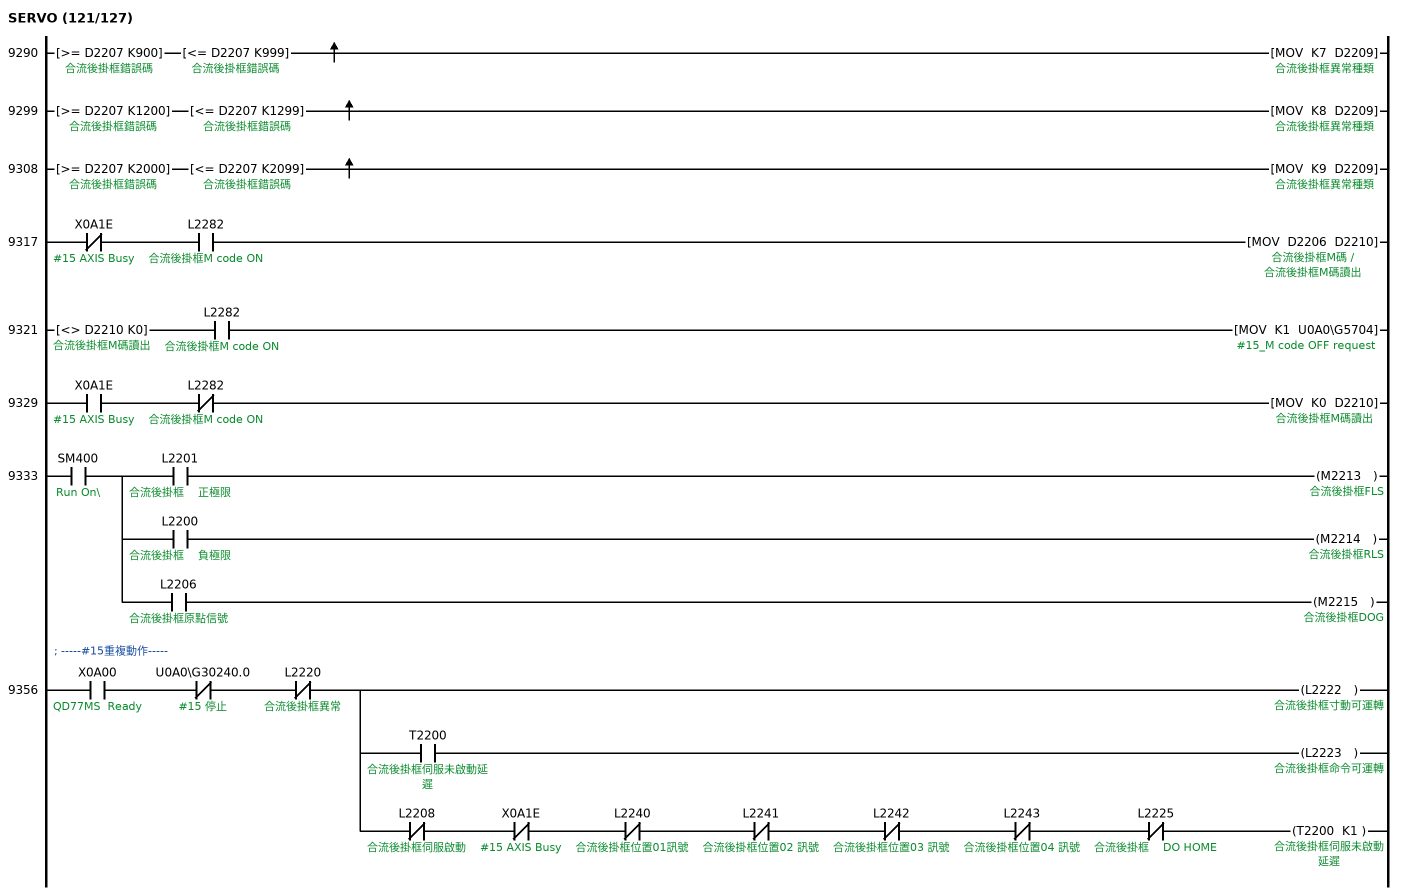
[picture p120: ladder of SERVO, rungs at steps 9290 to 9356]
9290  LD>=    D2207 K900  ; 合流後掛框錯誤碼
      AND<=   D2207 K999  ; 合流後掛框錯誤碼
      MEP
      MOV     K7 D2209
9299  LD>=    D2207 K1200  ; 合流後掛框錯誤碼
      AND<=   D2207 K1299  ; 合流後掛框錯誤碼
      MEP
      MOV     K8 D2209
9308  LD>=    D2207 K2000  ; 合流後掛框錯誤碼
      AND<=   D2207 K2099  ; 合流後掛框錯誤碼
      MEP
      MOV     K9 D2209
9317  LDI     X0A1E  ; #15 AXIS Busy
      AND     L2282  ; 合流後掛框M code ON
      MOV     D2206 D2210  ; 合流後掛框M碼讀出
9321  LD<>    D2210 K0  ; 合流後掛框M碼讀出
      AND     L2282  ; 合流後掛框M code ON
      MOV     K1 U0A0\G5704  ; #15_M code OFF request
9329  LD      X0A1E  ; #15 AXIS Busy
      ANI     L2282  ; 合流後掛框M code ON
      MOV     K0 D2210
9333  LD      SM400  ; Run On\
      MPS
      AND     L2201  ; 合流後掛框    正極限
      OUT     M2213  ; 合流後掛框FLS
      MRD
      AND     L2200  ; 合流後掛框    負極限
      OUT     M2214  ; 合流後掛框RLS
      MPP
      AND     L2206  ; 合流後掛框原點信號
      OUT     M2215  ; 合流後掛框DOG
; -----#15重複動作-----
9356  LD      X0A00  ; QD77MS  Ready
      ANI     U0A0\G30240.0  ; #15 停止
      ANI     L2220  ; 合流後掛框異常
      OUT     L2222  ; 合流後掛框寸動可運轉
      MPS
      AND     T2200  ; 合流後掛框伺服未啟動延遲
      OUT     L2223  ; 合流後掛框命令可運轉
      MPP
      ANI     L2208  ; 合流後掛框伺服啟動
      ANI     X0A1E  ; #15 AXIS Busy
      ANI     L2240  ; 合流後掛框位置01訊號
      ANI     L2241  ; 合流後掛框位置02 訊號
      ANI     L2242  ; 合流後掛框位置03 訊號
      ANI     L2243  ; 合流後掛框位置04 訊號
      ANI     L2225  ; 合流後掛框    DO HOME
      OUT     T2200 K1  ; 合流後掛框伺服未啟動延遲
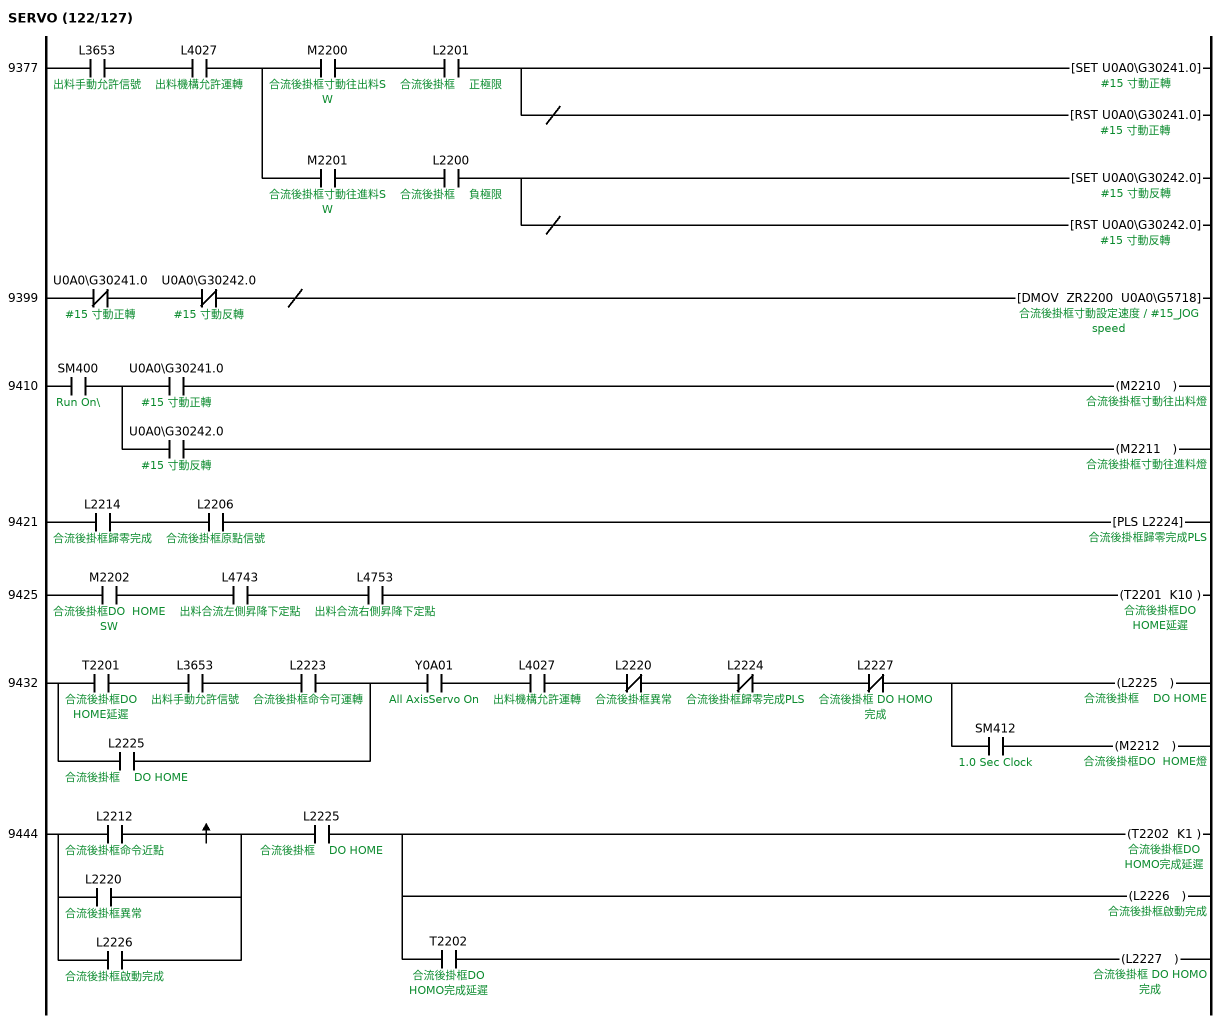
9377  LD      L3653  ; 出料手動允許信號
      AND     L4027  ; 出料機構允許運轉
      MPS
      AND     M2200  ; 合流後掛框寸動往出料SW
      AND     L2201  ; 合流後掛框    正極限
      SET     U0A0\G30241.0  ; #15 寸動正轉
      INV
      RST     U0A0\G30241.0  ; #15 寸動正轉
      MPP
      AND     M2201  ; 合流後掛框寸動往進料SW
      AND     L2200  ; 合流後掛框    負極限
      SET     U0A0\G30242.0  ; #15 寸動反轉
      INV
      RST     U0A0\G30242.0  ; #15 寸動反轉
9399  LDI     U0A0\G30241.0  ; #15 寸動正轉
      ANI     U0A0\G30242.0  ; #15 寸動反轉
      INV
      DMOV    ZR2200 U0A0\G5718  ; 合流後掛框寸動設定速度 / #15_JOG     speed
9410  LD      SM400  ; Run On\
      MPS
      AND     U0A0\G30241.0  ; #15 寸動正轉
      OUT     M2210  ; 合流後掛框寸動往出料燈
      MPP
      AND     U0A0\G30242.0  ; #15 寸動反轉
      OUT     M2211  ; 合流後掛框寸動往進料燈
9421  LD      L2214  ; 合流後掛框歸零完成
      AND     L2206  ; 合流後掛框原點信號
      PLS     L2224  ; 合流後掛框歸零完成PLS
9425  LD      M2202  ; 合流後掛框DO  HOME SW
      AND     L4743  ; 出料合流左側昇降下定點
      AND     L4753  ; 出料合流右側昇降下定點
      OUT     T2201 K10  ; 合流後掛框DO HOME延遲
9432  LD      T2201  ; 合流後掛框DO HOME延遲
      AND     L3653  ; 出料手動允許信號
      AND     L2223  ; 合流後掛框命令可運轉
      OR      L2225  ; 合流後掛框    DO HOME
      AND     Y0A01  ; All AxisServo On
      AND     L4027  ; 出料機構允許運轉
      ANI     L2220  ; 合流後掛框異常
      ANI     L2224  ; 合流後掛框歸零完成PLS
      ANI     L2227  ; 合流後掛框 DO HOMO 完成
      OUT     L2225  ; 合流後掛框    DO HOME
      AND     SM412  ; 1.0 Sec Clock
      OUT     M2212  ; 合流後掛框DO  HOME燈
9444  LD      L2212  ; 合流後掛框命令近點
      MEP
      OR      L2220  ; 合流後掛框異常
      OR      L2226  ; 合流後掛框啟動完成
      AND     L2225  ; 合流後掛框    DO HOME
      OUT     T2202 K1  ; 合流後掛框DO HOMO完成延遲
      OUT     L2226  ; 合流後掛框啟動完成
      AND     T2202  ; 合流後掛框DO HOMO完成延遲
      OUT     L2227  ; 合流後掛框 DO HOMO 完成
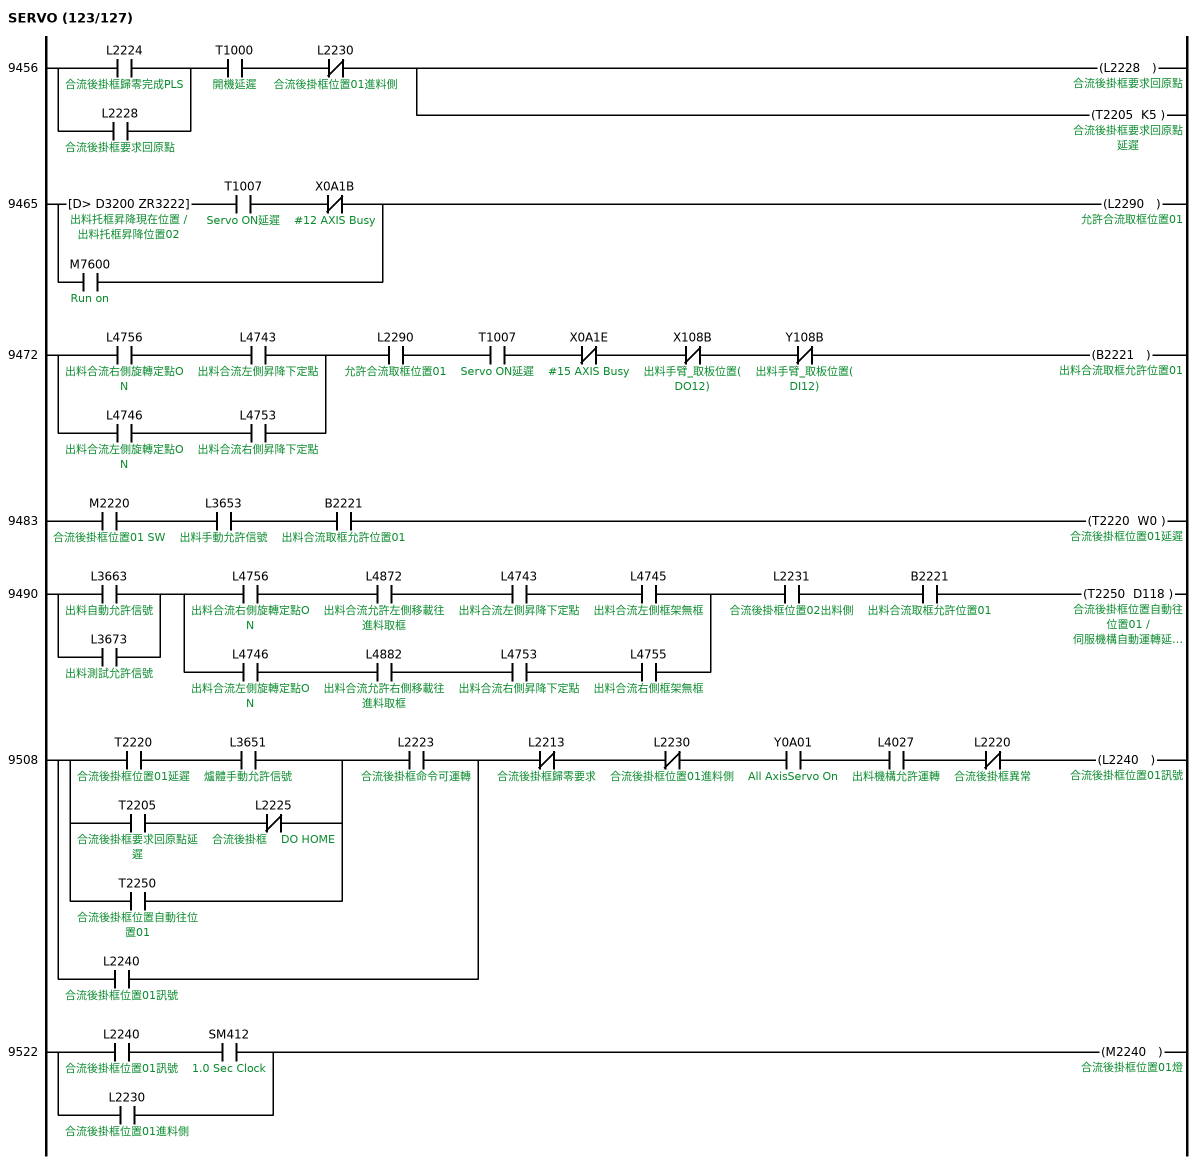
9456  LD      L2224  ; 合流後掛框歸零完成PLS
      OR      L2228  ; 合流後掛框要求回原點
      AND     T1000  ; 開機延遲
      ANI     L2230  ; 合流後掛框位置01進料側
      OUT     L2228  ; 合流後掛框要求回原點
      OUT     T2205 K5  ; 合流後掛框要求回原點延遲
9465  LDD>    D3200 ZR3222  ; 出料托框昇降現在位置 / 出料托框昇降位置02
      AND     T1007  ; Servo ON延遲
      ANI     X0A1B  ; #12 AXIS Busy
      OR      M7600  ; Run on
      OUT     L2290  ; 允許合流取框位置01
9472  LD      L4756  ; 出料合流右側旋轉定點ON
      AND     L4743  ; 出料合流左側昇降下定點
      LD      L4746  ; 出料合流左側旋轉定點ON
      AND     L4753  ; 出料合流右側昇降下定點
      ORB
      AND     L2290  ; 允許合流取框位置01
      AND     T1007  ; Servo ON延遲
      ANI     X0A1E  ; #15 AXIS Busy
      ANI     X108B  ; 出料手臂_取板位置(DO12)
      ANI     Y108B  ; 出料手臂_取板位置(DI12)
      OUT     B2221  ; 出料合流取框允許位置01
9483  LD      M2220  ; 合流後掛框位置01 SW
      AND     L3653  ; 出料手動允許信號
      AND     B2221  ; 出料合流取框允許位置01
      OUT     T2220 W0  ; 合流後掛框位置01延遲
9490  LD      L3663  ; 出料自動允許信號
      OR      L3673  ; 出料測試允許信號
      LD      L4756  ; 出料合流右側旋轉定點ON
      AND     L4872  ; 出料合流允許左側移載往  進料取框
      AND     L4743  ; 出料合流左側昇降下定點
      AND     L4745  ; 出料合流左側框架無框
      LD      L4746  ; 出料合流左側旋轉定點ON
      AND     L4882  ; 出料合流允許右側移載往  進料取框
      AND     L4753  ; 出料合流右側昇降下定點
      AND     L4755  ; 出料合流右側框架無框
      ORB
      ANB
      AND     L2231  ; 合流後掛框位置02出料側
      AND     B2221  ; 出料合流取框允許位置01
      OUT     T2250 D118  ; 合流後掛框位置自動往位置01 / 伺服機構自動運轉延遲時間
9508  LD      T2220  ; 合流後掛框位置01延遲
      AND     L3651  ; 爐體手動允許信號
      LD      T2205  ; 合流後掛框要求回原點延遲
      ANI     L2225  ; 合流後掛框    DO HOME
      ORB
      OR      T2250  ; 合流後掛框位置自動往位置01
      AND     L2223  ; 合流後掛框命令可運轉
      OR      L2240  ; 合流後掛框位置01訊號
      ANI     L2213  ; 合流後掛框歸零要求
      ANI     L2230  ; 合流後掛框位置01進料側
      AND     Y0A01  ; All AxisServo On
      AND     L4027  ; 出料機構允許運轉
      ANI     L2220  ; 合流後掛框異常
      OUT     L2240  ; 合流後掛框位置01訊號
9522  LD      L2240  ; 合流後掛框位置01訊號
      AND     SM412  ; 1.0 Sec Clock
      OR      L2230  ; 合流後掛框位置01進料側
      OUT     M2240  ; 合流後掛框位置01燈
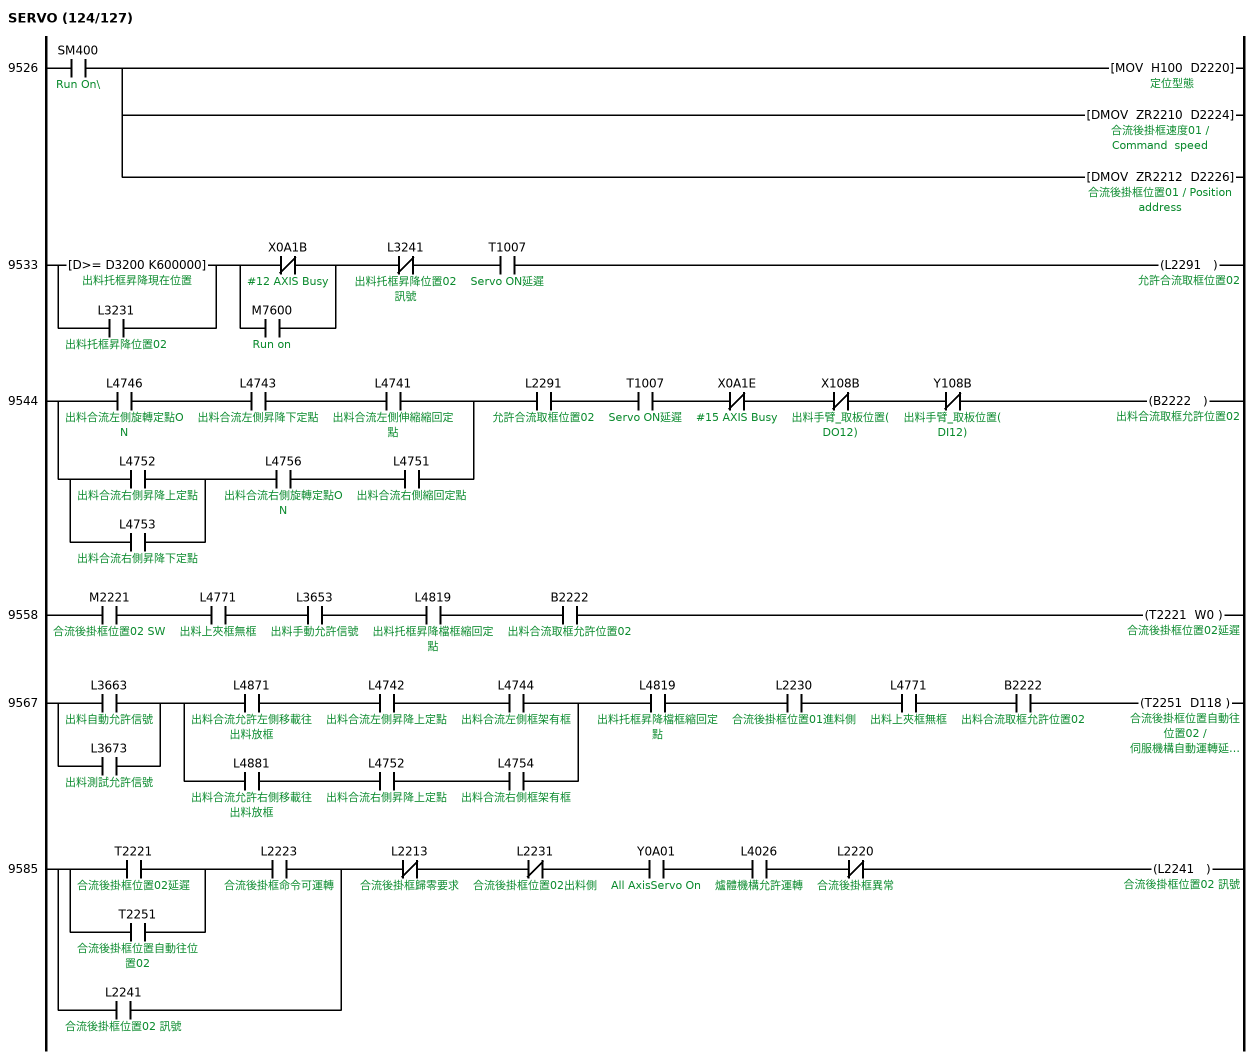
9526  LD      SM400  ; Run On\
      MOV     H100 D2220  ; 定位型態
      DMOV    ZR2210 D2224  ; 合流後掛框速度01 / Command  speed
      DMOV    ZR2212 D2226  ; Position address
9533  LDD>=   D3200 K600000  ; 出料托框昇降現在位置
      OR      L3231  ; 出料托框昇降位置02
      LDI     X0A1B  ; #12 AXIS Busy
      OR      M7600  ; Run on
      ANB
      ANI     L3241  ; 出料托框昇降位置02 訊號
      AND     T1007  ; Servo ON延遲
      OUT     L2291  ; 允許合流取框位置02
9544  LD      L4746  ; 出料合流左側旋轉定點ON
      AND     L4743  ; 出料合流左側昇降下定點
      AND     L4741  ; 出料合流左側伸縮縮回定點
      LD      L4752  ; 出料合流右側昇降上定點
      OR      L4753  ; 出料合流右側昇降下定點
      AND     L4756  ; 出料合流右側旋轉定點ON
      AND     L4751  ; 出料合流右側縮回定點
      ORB
      AND     L2291  ; 允許合流取框位置02
      AND     T1007  ; Servo ON延遲
      ANI     X0A1E  ; #15 AXIS Busy
      ANI     X108B  ; 出料手臂_取板位置(DO12)
      ANI     Y108B  ; 出料手臂_取板位置(DI12)
      OUT     B2222  ; 出料合流取框允許位置02
9558  LD      M2221  ; 合流後掛框位置02 SW
      AND     L4771  ; 出料上夾框無框
      AND     L3653  ; 出料手動允許信號
      AND     L4819  ; 出料托框昇降檔框縮回定點
      AND     B2222  ; 出料合流取框允許位置02
      OUT     T2221 W0  ; 合流後掛框位置02延遲
9567  LD      L3663  ; 出料自動允許信號
      OR      L3673  ; 出料測試允許信號
      LD      L4871  ; 出料合流允許左側移載往  出料放框
      AND     L4742  ; 出料合流左側昇降上定點
      AND     L4744  ; 出料合流左側框架有框
      LD      L4881  ; 出料合流允許右側移載往  出料放框
      AND     L4752  ; 出料合流右側昇降上定點
      AND     L4754  ; 出料合流右側框架有框
      ORB
      ANB
      AND     L4819  ; 出料托框昇降檔框縮回定點
      AND     L2230  ; 合流後掛框位置01進料側
      AND     L4771  ; 出料上夾框無框
      AND     B2222  ; 出料合流取框允許位置02
      OUT     T2251 D118  ; 合流後掛框位置自動往位置02 / 伺服機構自動運轉延遲時間
9585  LD      T2221  ; 合流後掛框位置02延遲
      OR      T2251  ; 合流後掛框位置自動往位置02
      AND     L2223  ; 合流後掛框命令可運轉
      OR      L2241  ; 合流後掛框位置02 訊號
      ANI     L2213  ; 合流後掛框歸零要求
      ANI     L2231  ; 合流後掛框位置02出料側
      AND     Y0A01  ; All AxisServo On
      AND     L4026  ; 爐體機構允許運轉
      ANI     L2220  ; 合流後掛框異常
      OUT     L2241  ; 合流後掛框位置02 訊號
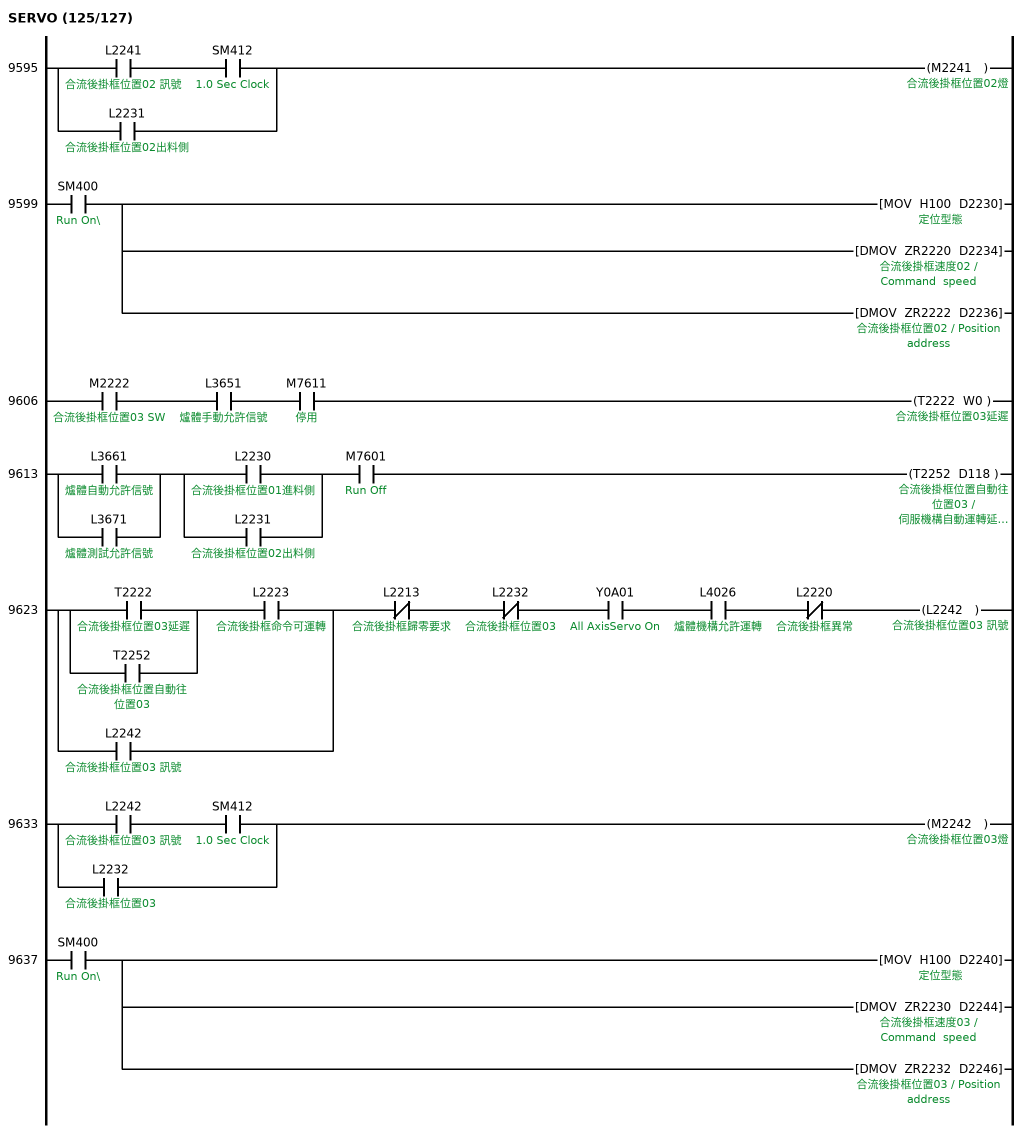
9595  LD      L2241  ; 合流後掛框位置02 訊號
      AND     SM412  ; 1.0 Sec Clock
      OR      L2231  ; 合流後掛框位置02出料側
      OUT     M2241  ; 合流後掛框位置02燈
9599  LD      SM400  ; Run On\
      MOV     H100 D2230  ; 定位型態
      DMOV    ZR2220 D2234  ; 合流後掛框速度02 / Command  speed
      DMOV    ZR2222 D2236  ; Position address
9606  LD      M2222  ; 合流後掛框位置03 SW
      AND     L3651  ; 爐體手動允許信號
      AND     M7611  ; 停用
      OUT     T2222 W0  ; 合流後掛框位置03延遲
9613  LD      L3661  ; 爐體自動允許信號
      OR      L3671  ; 爐體測試允許信號
      LD      L2230  ; 合流後掛框位置01進料側
      OR      L2231  ; 合流後掛框位置02出料側
      ANB
      AND     M7601  ; Run Off
      OUT     T2252 D118  ; 合流後掛框位置自動往  位置03 / 伺服機構自動運轉延遲時間
9623  LD      T2222  ; 合流後掛框位置03延遲
      OR      T2252  ; 合流後掛框位置自動往  位置03
      AND     L2223  ; 合流後掛框命令可運轉
      OR      L2242  ; 合流後掛框位置03 訊號
      ANI     L2213  ; 合流後掛框歸零要求
      ANI     L2232  ; 合流後掛框位置03
      AND     Y0A01  ; All AxisServo On
      AND     L4026  ; 爐體機構允許運轉
      ANI     L2220  ; 合流後掛框異常
      OUT     L2242  ; 合流後掛框位置03 訊號
9633  LD      L2242  ; 合流後掛框位置03 訊號
      AND     SM412  ; 1.0 Sec Clock
      OR      L2232  ; 合流後掛框位置03
      OUT     M2242  ; 合流後掛框位置03燈
9637  LD      SM400  ; Run On\
      MOV     H100 D2240  ; 定位型態
      DMOV    ZR2230 D2244  ; 合流後掛框速度03 / Command  speed
      DMOV    ZR2232 D2246  ; Position address
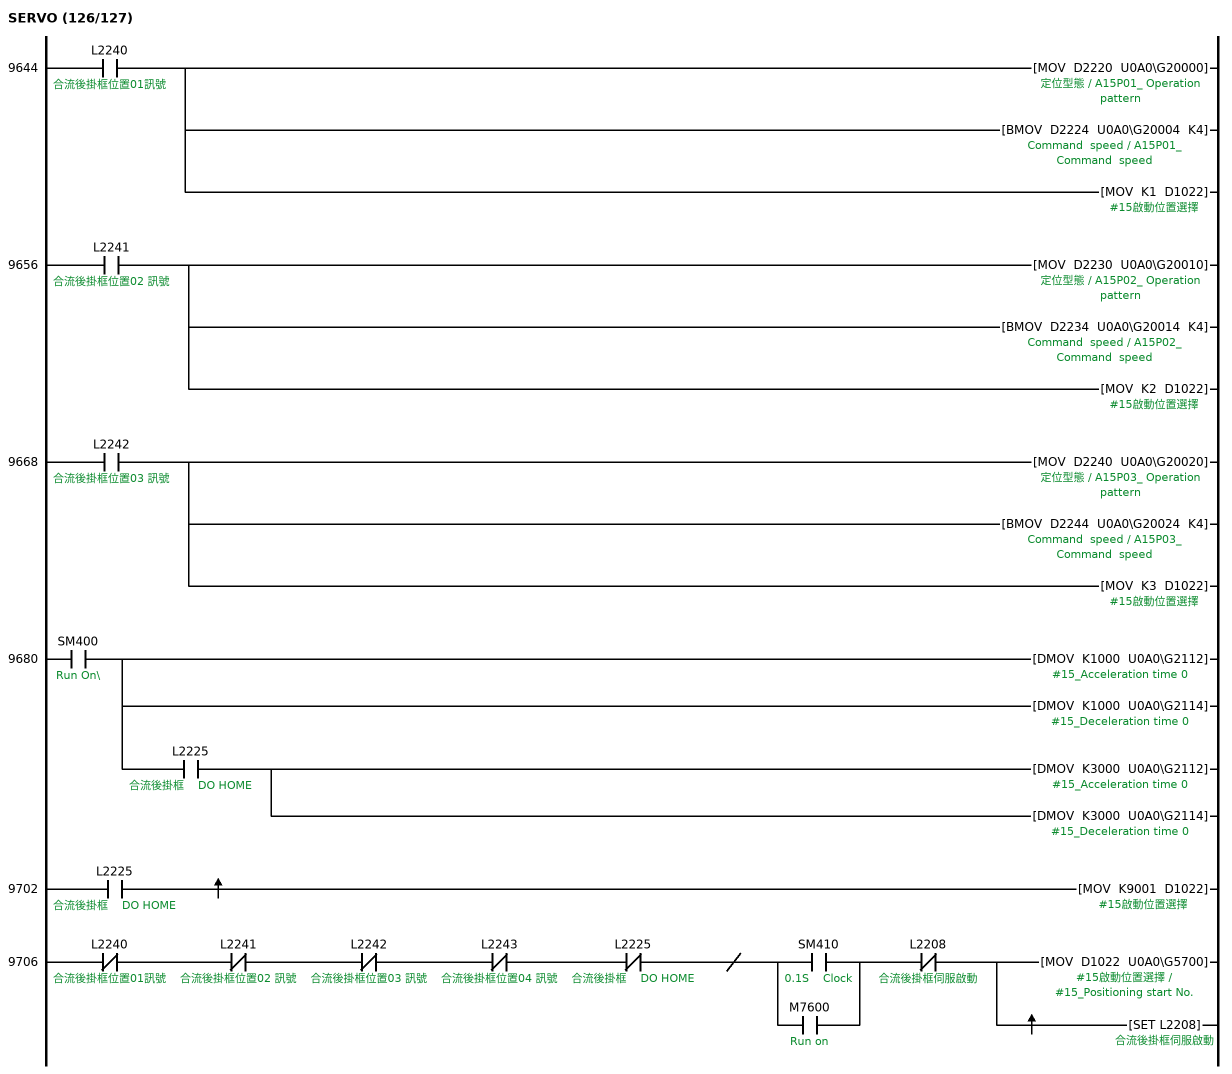
9644  LD      L2240  ; 合流後掛框位置01訊號
      MOV     D2220 U0A0\G20000  ; A15P01_ Operation pattern
      BMOV    D2224 U0A0\G20004 K4  ; A15P01_ Command  speed
      MOV     K1 D1022  ; #15啟動位置選擇
9656  LD      L2241  ; 合流後掛框位置02 訊號
      MOV     D2230 U0A0\G20010  ; A15P02_ Operation pattern
      BMOV    D2234 U0A0\G20014 K4  ; A15P02_ Command  speed
      MOV     K2 D1022
9668  LD      L2242  ; 合流後掛框位置03 訊號
      MOV     D2240 U0A0\G20020  ; A15P03_ Operation pattern
      BMOV    D2244 U0A0\G20024 K4  ; A15P03_ Command  speed
      MOV     K3 D1022
9680  LD      SM400  ; Run On\
      DMOV    K1000 U0A0\G2112  ; #15_Acceleration time 0
      DMOV    K1000 U0A0\G2114  ; #15_Deceleration time 0
      AND     L2225  ; 合流後掛框    DO HOME
      DMOV    K3000 U0A0\G2112
      DMOV    K3000 U0A0\G2114
9702  LD      L2225  ; 合流後掛框    DO HOME
      MEP
      MOV     K9001 D1022
9706  LDI     L2240  ; 合流後掛框位置01訊號
      ANI     L2241  ; 合流後掛框位置02 訊號
      ANI     L2242  ; 合流後掛框位置03 訊號
      ANI     L2243  ; 合流後掛框位置04 訊號
      ANI     L2225  ; 合流後掛框    DO HOME
      INV
      LD      SM410  ; 0.1S    Clock
      OR      M7600  ; Run on
      ANB
      ANI     L2208  ; 合流後掛框伺服啟動
      MOV     D1022 U0A0\G5700  ; #15_Positioning start No.
      MEP
      SET     L2208  ; 合流後掛框伺服啟動
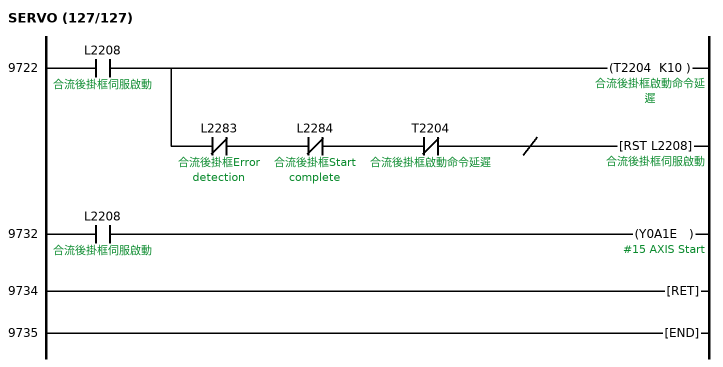
9722  LD      L2208  ; 合流後掛框伺服啟動
      OUT     T2204 K10  ; 合流後掛框啟動命令延遲
      ANI     L2283  ; 合流後掛框Error detection
      ANI     L2284  ; 合流後掛框Start complete
      ANI     T2204  ; 合流後掛框啟動命令延遲
      INV
      RST     L2208  ; 合流後掛框伺服啟動
9732  LD      L2208  ; 合流後掛框伺服啟動
      OUT     Y0A1E  ; #15 AXIS Start
9734  RET
9735  END
END_PROGRAM

PROGRAM MAIN
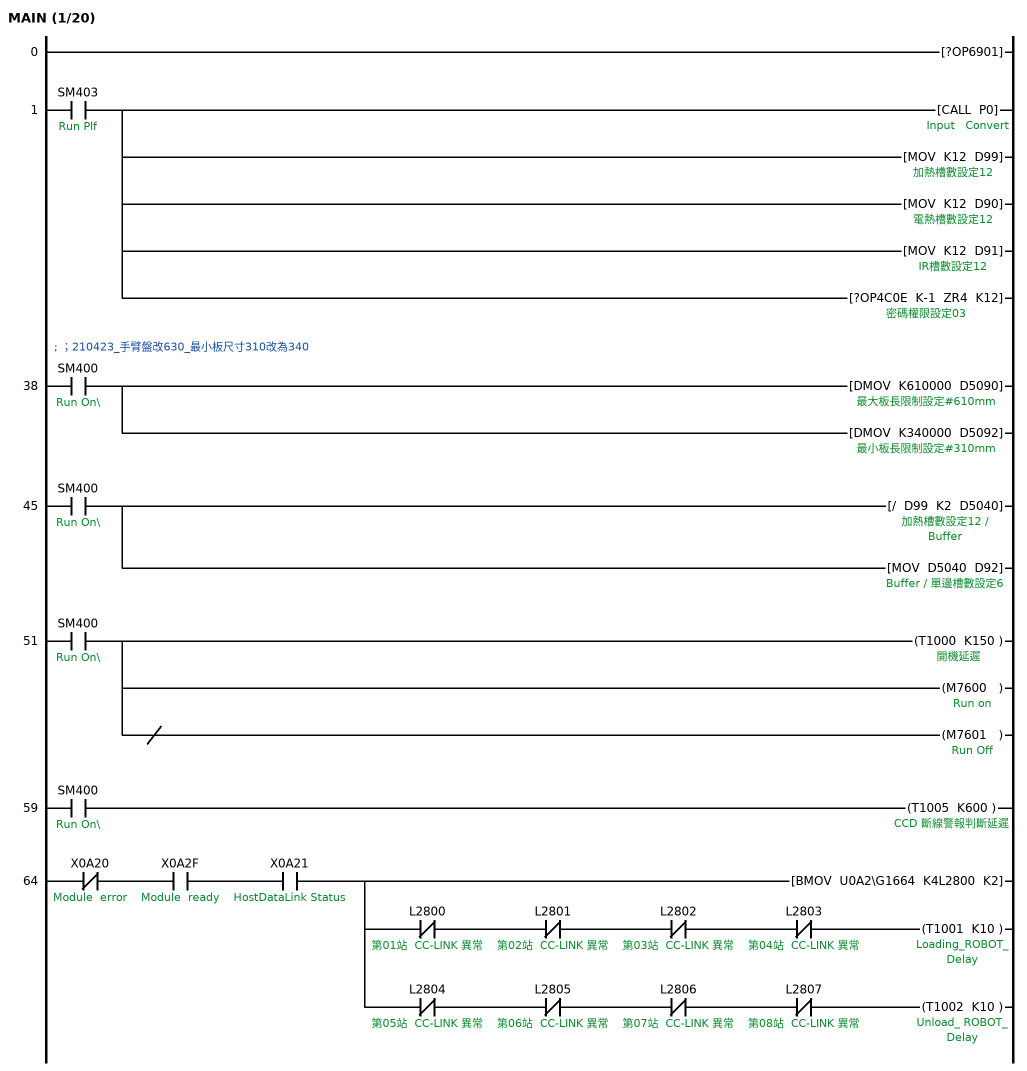
0     ?OP6901
1     LD      SM403  ; Run Plf
      CALL    P0  ; Input   Convert
      MOV     K12 D99  ; 加熱槽數設定12
      MOV     K12 D90  ; 電熱槽數設定12
      MOV     K12 D91  ; IR槽數設定12
      ?OP4C0E K-1 ZR4 K12  ; 密碼權限設定03
; ；210423_手臂盤改630_最小板尺寸310改為340
38    LD      SM400  ; Run On\
      DMOV    K610000 D5090  ; 最大板長限制設定#610mm
      DMOV    K340000 D5092  ; 最小板長限制設定#310mm
45    LD      SM400  ; Run On\
      /       D99 K2 D5040  ; Buffer
      MOV     D5040 D92  ; 單邊槽數設定6
51    LD      SM400  ; Run On\
      OUT     T1000 K150  ; 開機延遲
      OUT     M7600  ; Run on
      INV
      OUT     M7601  ; Run Off
59    LD      SM400  ; Run On\
      OUT     T1005 K600  ; CCD 斷線警報判斷延遲
64    LDI     X0A20  ; Module  error
      AND     X0A2F  ; Module  ready
      AND     X0A21  ; HostDataLink Status
      BMOV    U0A2\G1664 K4L2800 K2  ; 第01站  CC-LINK 異常
      MPS
      ANI     L2800  ; 第01站  CC-LINK 異常
      ANI     L2801  ; 第02站  CC-LINK 異常
      ANI     L2802  ; 第03站  CC-LINK 異常
      ANI     L2803  ; 第04站  CC-LINK 異常
      OUT     T1001 K10  ; Loading_ROBOT_  Delay
      MPP
      ANI     L2804  ; 第05站  CC-LINK 異常
      ANI     L2805  ; 第06站  CC-LINK 異常
      ANI     L2806  ; 第07站  CC-LINK 異常
      ANI     L2807  ; 第08站  CC-LINK 異常
      OUT     T1002 K10  ; Unload_ ROBOT_  Delay
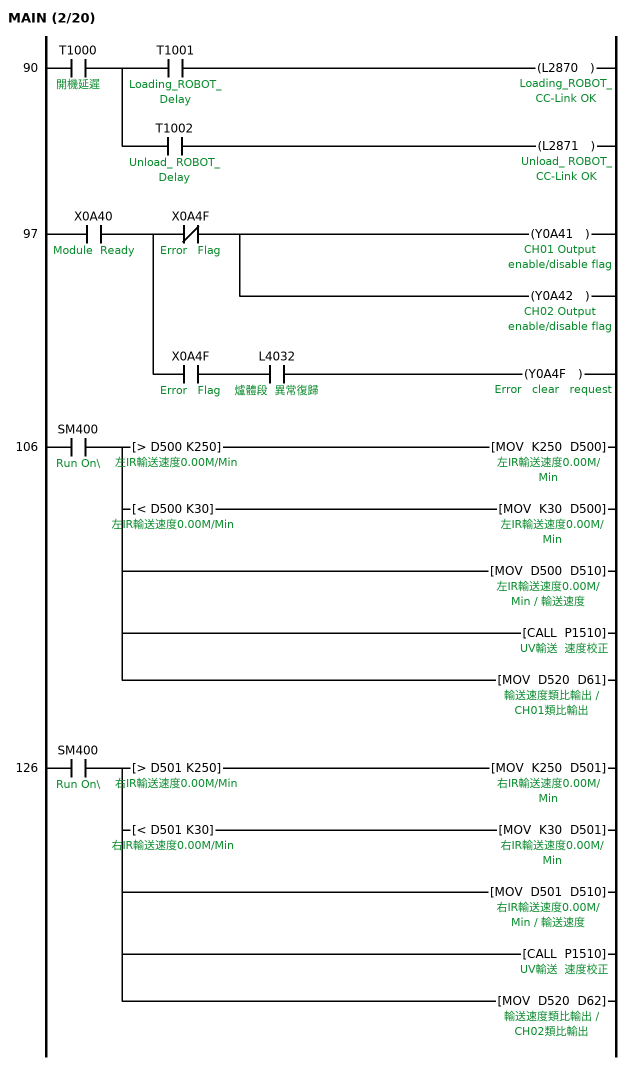
90    LD      T1000  ; 開機延遲
      MPS
      AND     T1001  ; Loading_ROBOT_  Delay
      OUT     L2870  ; Loading_ROBOT_  CC-Link OK
      MPP
      AND     T1002  ; Unload_ ROBOT_  Delay
      OUT     L2871  ; Unload_ ROBOT_  CC-Link OK
97    LD      X0A40  ; Module  Ready
      MPS
      ANI     X0A4F  ; Error   Flag
      OUT     Y0A41  ; CH01 Output enable/disable flag
      OUT     Y0A42  ; CH02 Output enable/disable flag
      MPP
      AND     X0A4F  ; Error   Flag
      AND     L4032  ; 爐體段  異常復歸
      OUT     Y0A4F  ; Error   clear   request
106   LD      SM400  ; Run On\
      MPS
      AND>    D500 K250  ; 左IR輸送速度0.00M/Min
      MOV     K250 D500
      MRD
      AND<    D500 K30  ; 左IR輸送速度0.00M/Min
      MOV     K30 D500
      MPP
      MOV     D500 D510  ; 輸送速度
      CALL    P1510  ; UV輸送  速度校正
      MOV     D520 D61  ; 輸送速度類比輸出 / CH01類比輸出
126   LD      SM400  ; Run On\
      MPS
      AND>    D501 K250  ; 右IR輸送速度0.00M/Min
      MOV     K250 D501
      MRD
      AND<    D501 K30  ; 右IR輸送速度0.00M/Min
      MOV     K30 D501
      MPP
      MOV     D501 D510
      CALL    P1510
      MOV     D520 D62  ; CH02類比輸出
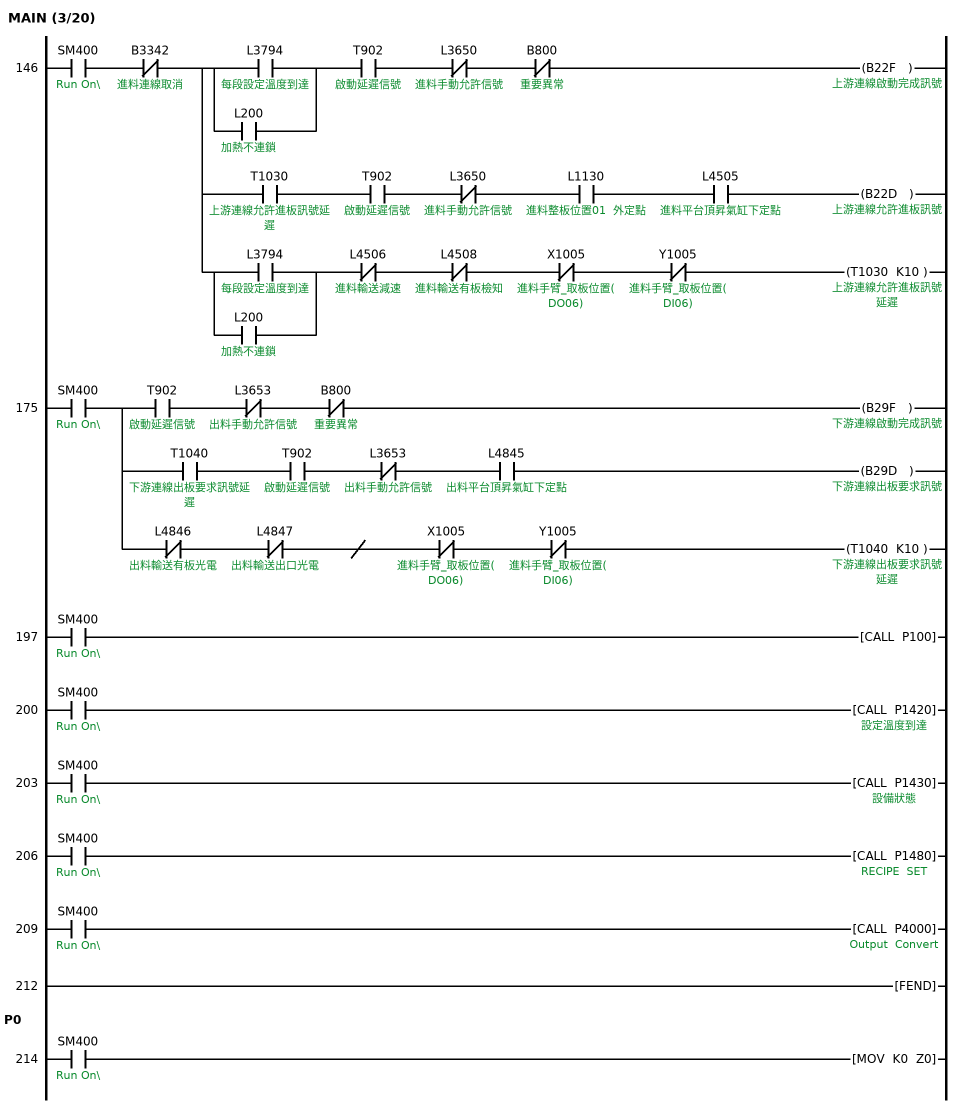
146   LD      SM400  ; Run On\
      ANI     B3342  ; 進料連線取消
      MPS
      LD      L3794  ; 每段設定溫度到達
      OR      L200  ; 加熱不連鎖
      ANB
      AND     T902  ; 啟動延遲信號
      ANI     L3650  ; 進料手動允許信號
      ANI     B800  ; 重要異常
      OUT     B22F  ; 上游連線啟動完成訊號
      MRD
      AND     T1030  ; 上游連線允許進板訊號延遲
      AND     T902  ; 啟動延遲信號
      ANI     L3650  ; 進料手動允許信號
      AND     L1130  ; 進料整板位置01  外定點
      AND     L4505  ; 進料平台頂昇氣缸下定點
      OUT     B22D  ; 上游連線允許進板訊號
      MPP
      LD      L3794  ; 每段設定溫度到達
      OR      L200  ; 加熱不連鎖
      ANB
      ANI     L4506  ; 進料輸送減速
      ANI     L4508  ; 進料輸送有板檢知
      ANI     X1005  ; 進料手臂_取板位置(DO06)
      ANI     Y1005  ; 進料手臂_取板位置(DI06)
      OUT     T1030 K10  ; 上游連線允許進板訊號延遲
175   LD      SM400  ; Run On\
      MPS
      AND     T902  ; 啟動延遲信號
      ANI     L3653  ; 出料手動允許信號
      ANI     B800  ; 重要異常
      OUT     B29F  ; 下游連線啟動完成訊號
      MRD
      AND     T1040  ; 下游連線出板要求訊號延遲
      AND     T902  ; 啟動延遲信號
      ANI     L3653  ; 出料手動允許信號
      AND     L4845  ; 出料平台頂昇氣缸下定點
      OUT     B29D  ; 下游連線出板要求訊號
      MPP
      ANI     L4846  ; 出料輸送有板光電
      ANI     L4847  ; 出料輸送出口光電
      INV
      ANI     X1005  ; 進料手臂_取板位置(DO06)
      ANI     Y1005  ; 進料手臂_取板位置(DI06)
      OUT     T1040 K10  ; 下游連線出板要求訊號延遲
197   LD      SM400  ; Run On\
      CALL    P100
200   LD      SM400  ; Run On\
      CALL    P1420  ; 設定溫度到達
203   LD      SM400  ; Run On\
      CALL    P1430  ; 設備狀態
206   LD      SM400  ; Run On\
      CALL    P1480  ; RECIPE  SET
209   LD      SM400  ; Run On\
      CALL    P4000  ; Output  Convert
212   FEND
      P0
214   LD      SM400  ; Run On\
      MOV     K0 Z0
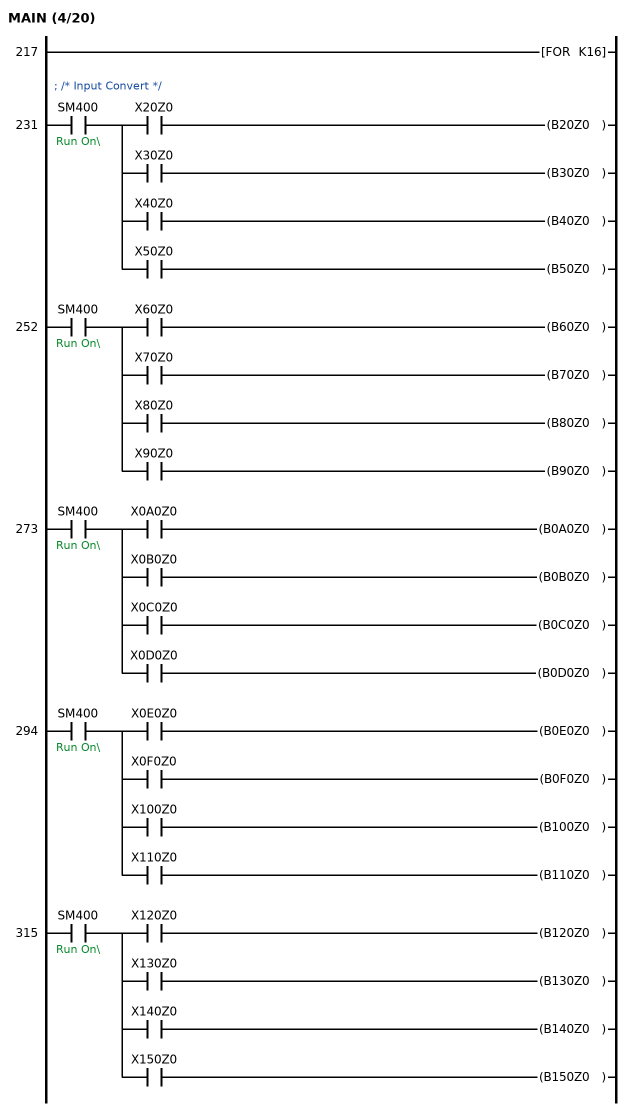
217   FOR     K16
; /* Input Convert */
231   LD      SM400  ; Run On\
      MPS
      AND     X20Z0
      OUT     B20Z0
      MRD
      AND     X30Z0
      OUT     B30Z0
      MRD
      AND     X40Z0
      OUT     B40Z0
      MPP
      AND     X50Z0
      OUT     B50Z0
252   LD      SM400  ; Run On\
      MPS
      AND     X60Z0
      OUT     B60Z0
      MRD
      AND     X70Z0
      OUT     B70Z0
      MRD
      AND     X80Z0
      OUT     B80Z0
      MPP
      AND     X90Z0
      OUT     B90Z0
273   LD      SM400  ; Run On\
      MPS
      AND     X0A0Z0
      OUT     B0A0Z0
      MRD
      AND     X0B0Z0
      OUT     B0B0Z0
      MRD
      AND     X0C0Z0
      OUT     B0C0Z0
      MPP
      AND     X0D0Z0
      OUT     B0D0Z0
294   LD      SM400  ; Run On\
      MPS
      AND     X0E0Z0
      OUT     B0E0Z0
      MRD
      AND     X0F0Z0
      OUT     B0F0Z0
      MRD
      AND     X100Z0
      OUT     B100Z0
      MPP
      AND     X110Z0
      OUT     B110Z0
315   LD      SM400  ; Run On\
      MPS
      AND     X120Z0
      OUT     B120Z0
      MRD
      AND     X130Z0
      OUT     B130Z0
      MRD
      AND     X140Z0
      OUT     B140Z0
      MPP
      AND     X150Z0
      OUT     B150Z0
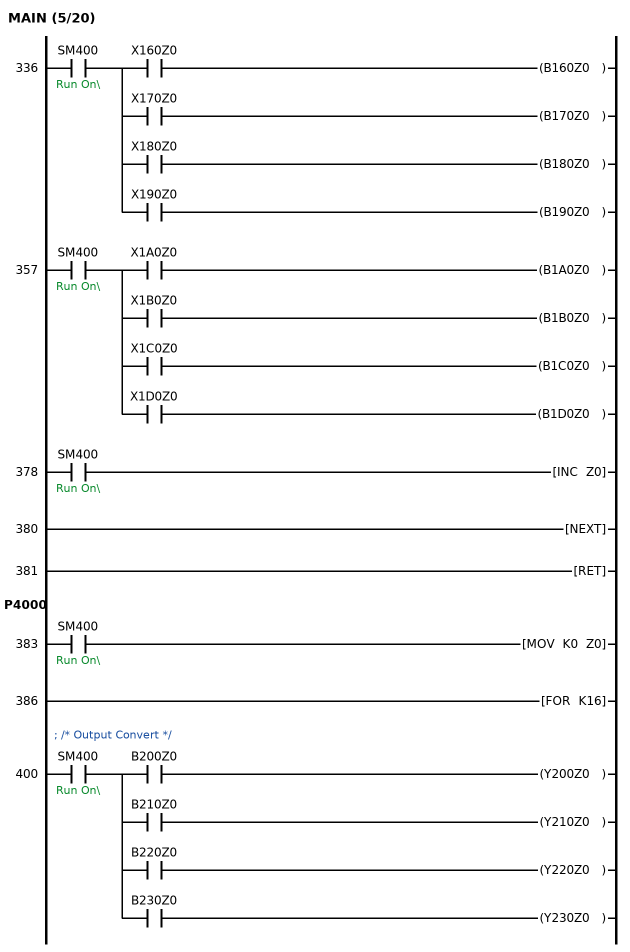
336   LD      SM400  ; Run On\
      MPS
      AND     X160Z0
      OUT     B160Z0
      MRD
      AND     X170Z0
      OUT     B170Z0
      MRD
      AND     X180Z0
      OUT     B180Z0
      MPP
      AND     X190Z0
      OUT     B190Z0
357   LD      SM400  ; Run On\
      MPS
      AND     X1A0Z0
      OUT     B1A0Z0
      MRD
      AND     X1B0Z0
      OUT     B1B0Z0
      MRD
      AND     X1C0Z0
      OUT     B1C0Z0
      MPP
      AND     X1D0Z0
      OUT     B1D0Z0
378   LD      SM400  ; Run On\
      INC     Z0
380   NEXT
381   RET
      P4000
383   LD      SM400  ; Run On\
      MOV     K0 Z0
386   FOR     K16
; /* Output Convert */
400   LD      SM400  ; Run On\
      MPS
      AND     B200Z0
      OUT     Y200Z0
      MRD
      AND     B210Z0
      OUT     Y210Z0
      MRD
      AND     B220Z0
      OUT     Y220Z0
      MPP
      AND     B230Z0
      OUT     Y230Z0
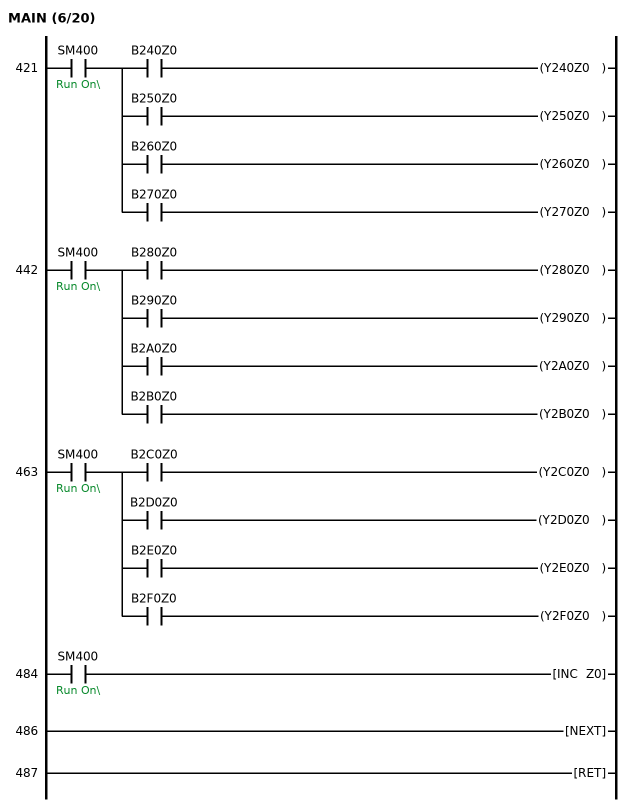
421   LD      SM400  ; Run On\
      MPS
      AND     B240Z0
      OUT     Y240Z0
      MRD
      AND     B250Z0
      OUT     Y250Z0
      MRD
      AND     B260Z0
      OUT     Y260Z0
      MPP
      AND     B270Z0
      OUT     Y270Z0
442   LD      SM400  ; Run On\
      MPS
      AND     B280Z0
      OUT     Y280Z0
      MRD
      AND     B290Z0
      OUT     Y290Z0
      MRD
      AND     B2A0Z0
      OUT     Y2A0Z0
      MPP
      AND     B2B0Z0
      OUT     Y2B0Z0
463   LD      SM400  ; Run On\
      MPS
      AND     B2C0Z0
      OUT     Y2C0Z0
      MRD
      AND     B2D0Z0
      OUT     Y2D0Z0
      MRD
      AND     B2E0Z0
      OUT     Y2E0Z0
      MPP
      AND     B2F0Z0
      OUT     Y2F0Z0
484   LD      SM400  ; Run On\
      INC     Z0
486   NEXT
487   RET
      P100
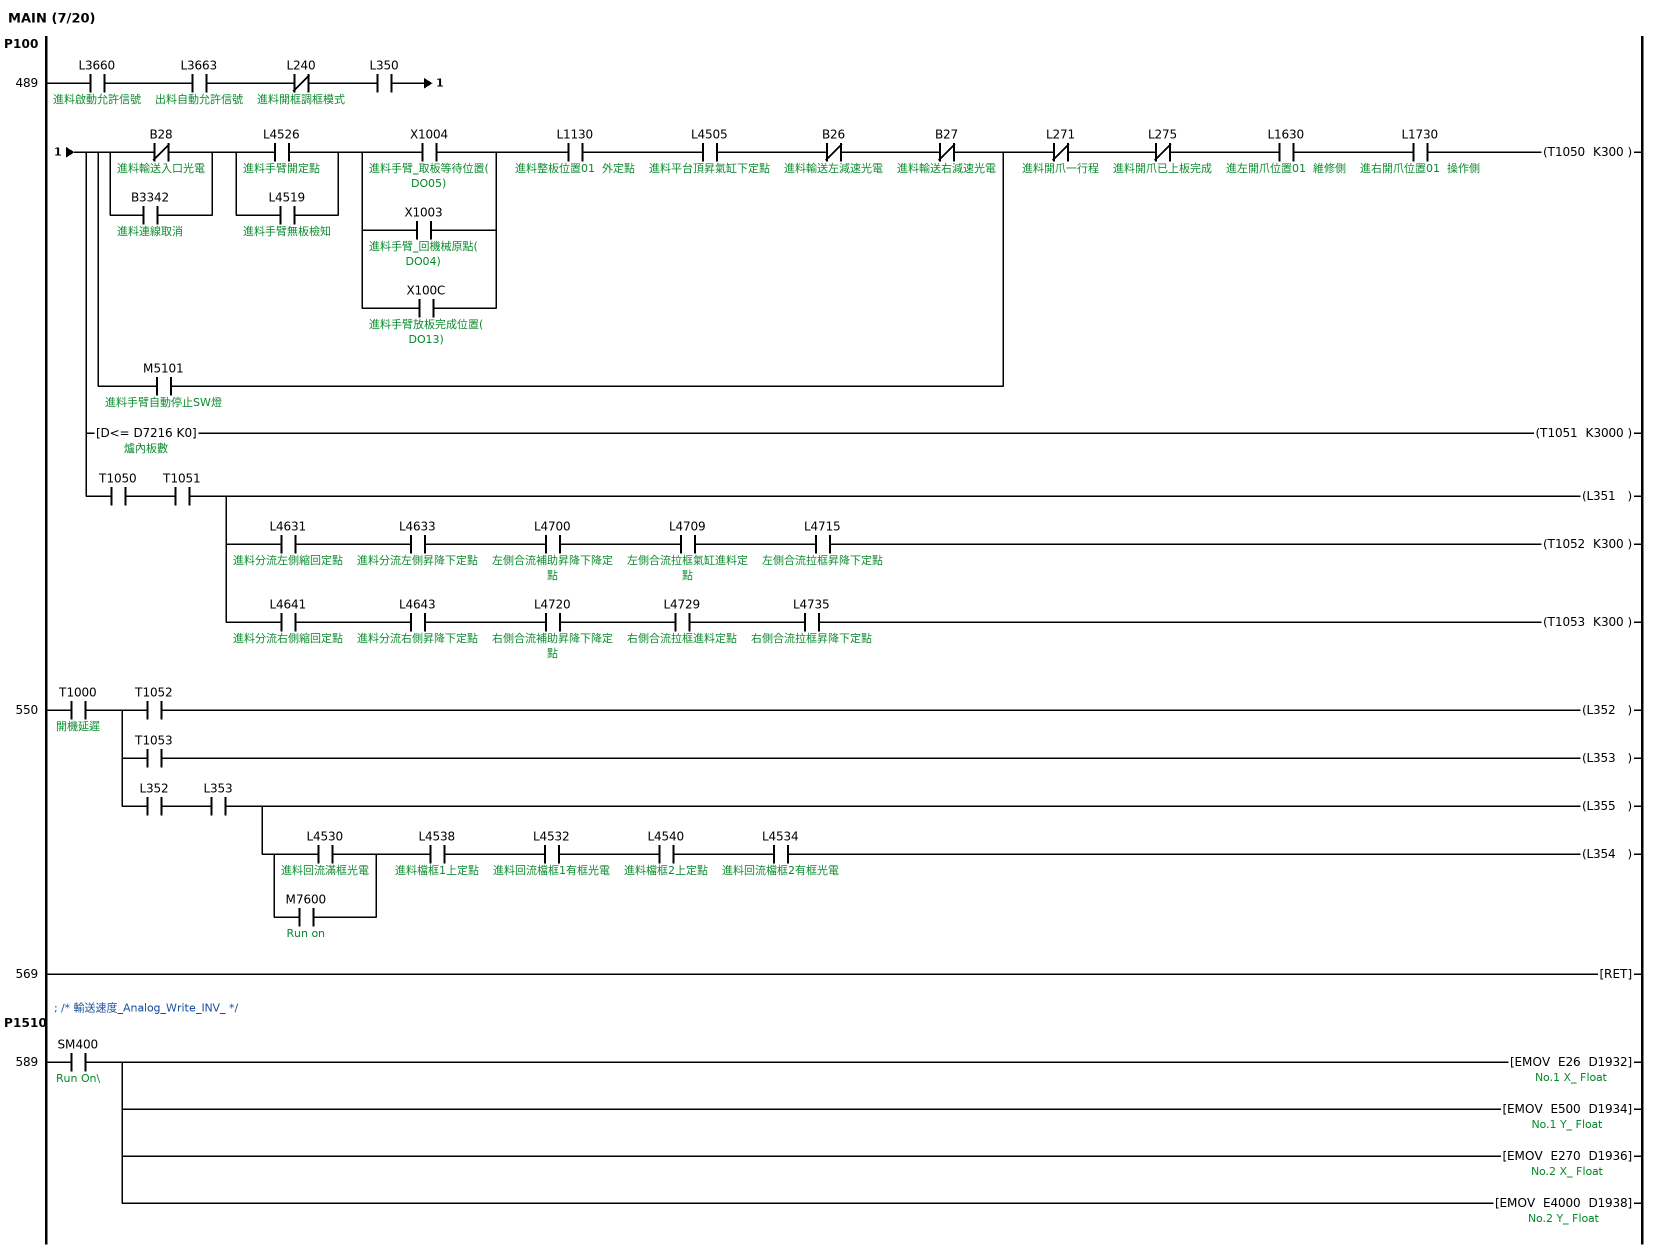
489   LD      L3660  ; 進料啟動允許信號
      AND     L3663  ; 出料自動允許信號
      ANI     L240  ; 進料開框調框模式
      AND     L350
      MPS
      LDI     B28  ; 進料輸送入口光電
      OR      B3342  ; 進料連線取消
      LD      L4526  ; 進料手臂開定點
      OR      L4519  ; 進料手臂無板檢知
      ANB
      LD      X1004  ; 進料手臂_取板等待位置(DO05)
      OR      X1003  ; 進料手臂_回機械原點(DO04)
      OR      X100C  ; 進料手臂放板完成位置(DO13)
      ANB
      AND     L1130  ; 進料整板位置01  外定點
      AND     L4505  ; 進料平台頂昇氣缸下定點
      ANI     B26  ; 進料輸送左減速光電
      ANI     B27  ; 進料輸送右減速光電
      OR      M5101  ; 進料手臂自動停止SW燈
      ANB
      ANI     L271  ; 進料開爪一行程
      ANI     L275  ; 進料開爪已上板完成
      AND     L1630  ; 進左開爪位置01  維修側
      AND     L1730  ; 進右開爪位置01  操作側
      OUT     T1050 K300
      MRD
      ANDD<=  D7216 K0  ; 爐內板數
      OUT     T1051 K3000
      MPP
      AND     T1050
      AND     T1051
      OUT     L351
      MPS
      AND     L4631  ; 進料分流左側縮回定點
      AND     L4633  ; 進料分流左側昇降下定點
      AND     L4700  ; 左側合流補助昇降下降定點
      AND     L4709  ; 左側合流拉框氣缸進料定點
      AND     L4715  ; 左側合流拉框昇降下定點
      OUT     T1052 K300
      MPP
      AND     L4641  ; 進料分流右側縮回定點
      AND     L4643  ; 進料分流右側昇降下定點
      AND     L4720  ; 右側合流補助昇降下降定點
      AND     L4729  ; 右側合流拉框進料定點
      AND     L4735  ; 右側合流拉框昇降下定點
      OUT     T1053 K300
550   LD      T1000  ; 開機延遲
      MPS
      AND     T1052
      OUT     L352
      MRD
      AND     T1053
      OUT     L353
      MPP
      AND     L352
      AND     L353
      OUT     L355
      LD      L4530  ; 進料回流滿框光電
      OR      M7600  ; Run on
      ANB
      AND     L4538  ; 進料檔框1上定點
      AND     L4532  ; 進料回流檔框1有框光電
      AND     L4540  ; 進料檔框2上定點
      AND     L4534  ; 進料回流檔框2有框光電
      OUT     L354
569   RET
      P1510
; /* 輸送速度_Analog_Write_INV_ */
589   LD      SM400  ; Run On\
      EMOV    E26 D1932  ; No.1 X_ Float
        [note] /* 類比值#500時_線速為_0.26M */
      EMOV    E500 D1934  ; No.1 Y_ Float
        [note] /* 類比值#500時_線速為_0.26M */
      EMOV    E270 D1936  ; No.2 X_ Float
        [note] /* 類比值#4000時_線速為_2.70M */
      EMOV    E4000 D1938  ; No.2 Y_ Float
        [note] /* 類比值#4000時_線速為_2.70M */
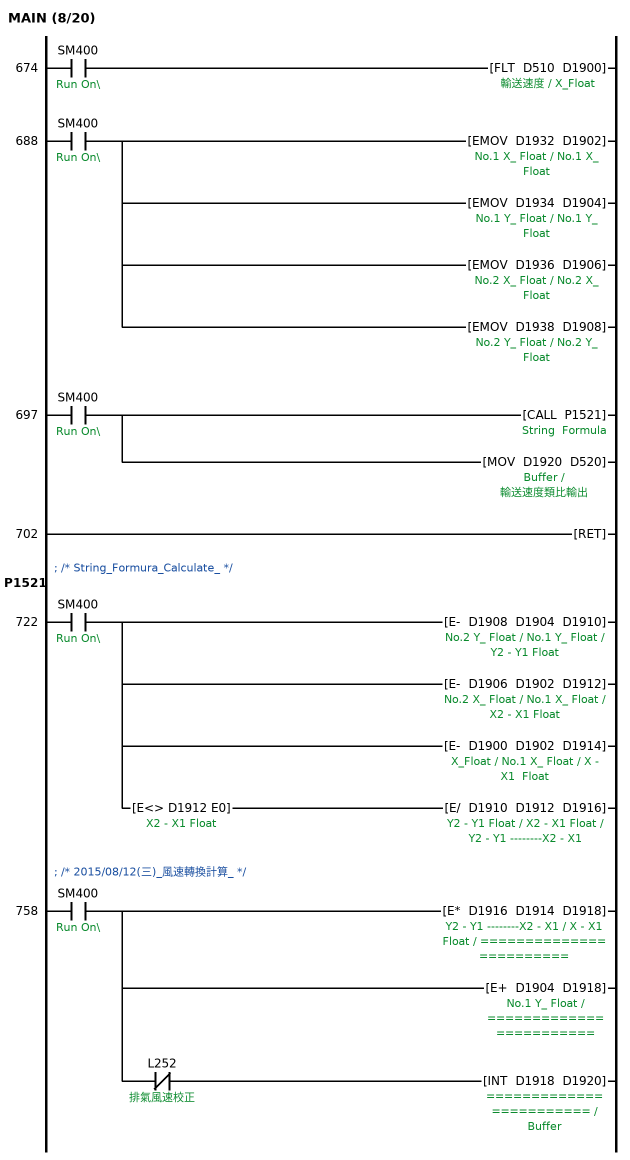
674   LD      SM400  ; Run On\
      FLT     D510 D1900  ; X_Float
        [note] /* 類比輸入值_ */
688   LD      SM400  ; Run On\
      EMOV    D1932 D1902  ; No.1 X_ Float
      EMOV    D1934 D1904  ; No.1 Y_ Float
      EMOV    D1936 D1906  ; No.2 X_ Float
      EMOV    D1938 D1908  ; No.2 Y_ Float
697   LD      SM400  ; Run On\
      CALL    P1521  ; String  Formula
      MOV     D1920 D520  ; Buffer
702   RET
      P1521
; /* String_Formura_Calculate_ */
722   LD      SM400  ; Run On\
      E-      D1908 D1904 D1910  ; Y2 - Y1 Float
      E-      D1906 D1902 D1912  ; X2 - X1 Float
      E-      D1900 D1902 D1914  ; X - X1  Float
      ANDE<>  D1912 E0  ; X2 - X1 Float
      E/      D1910 D1912 D1916  ; Y2 - Y1 --------X2 - X1
; /* 2015/08/12(三)_風速轉換計算_ */
758   LD      SM400  ; Run On\
      E*      D1916 D1914 D1918  ; ========================
      E+      D1904 D1918
      ANI     L252  ; 排氣風速校正
      INT     D1918 D1920
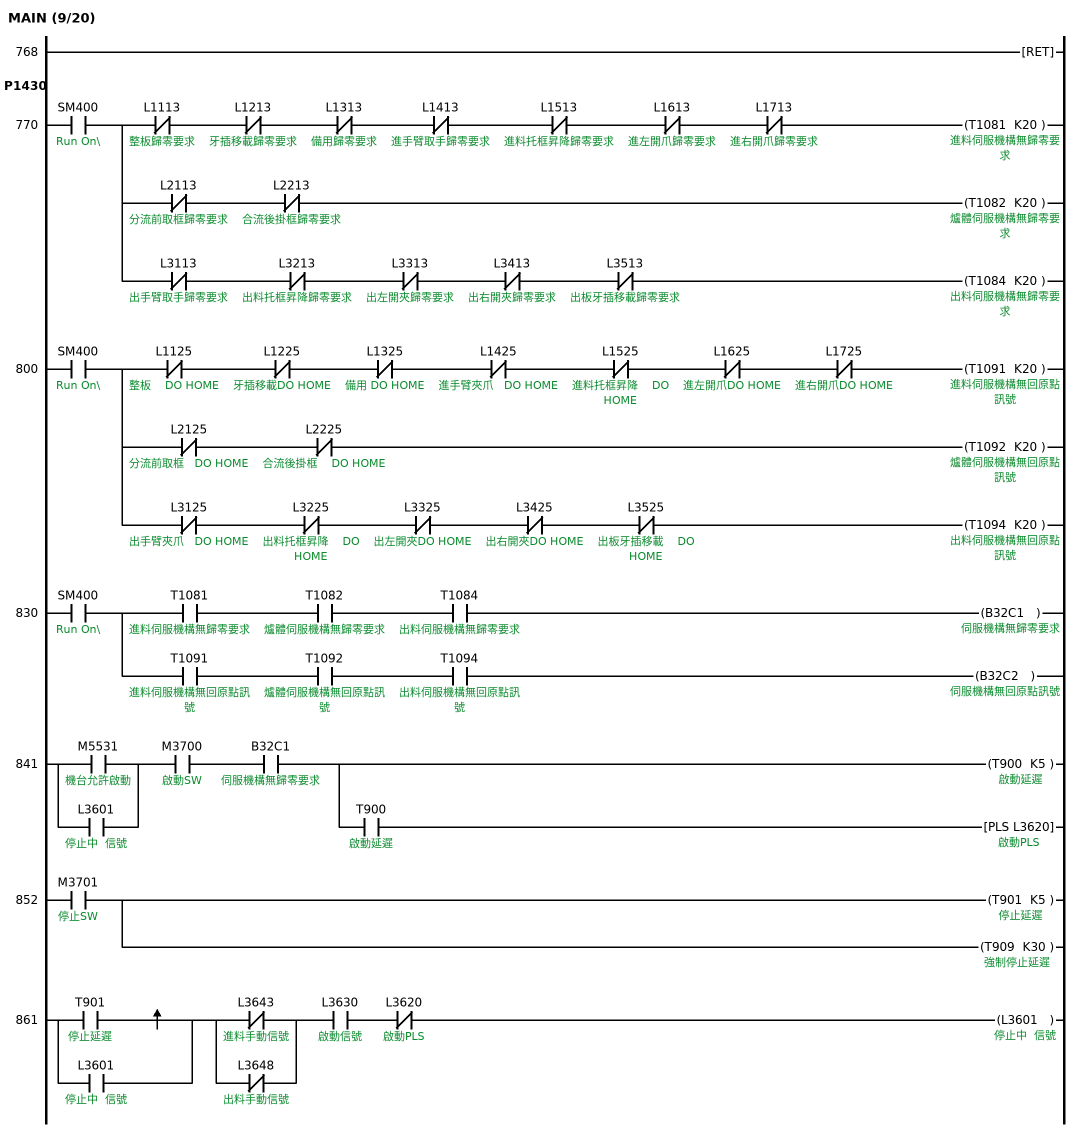
768   RET
      P1430
770   LD      SM400  ; Run On\
      MPS
      ANI     L1113  ; 整板歸零要求
      ANI     L1213  ; 牙插移載歸零要求
      ANI     L1313  ; 備用歸零要求
      ANI     L1413  ; 進手臂取手歸零要求
      ANI     L1513  ; 進料托框昇降歸零要求
      ANI     L1613  ; 進左開爪歸零要求
      ANI     L1713  ; 進右開爪歸零要求
      OUT     T1081 K20  ; 進料伺服機構無歸零要求
      MRD
      ANI     L2113  ; 分流前取框歸零要求
      ANI     L2213  ; 合流後掛框歸零要求
      OUT     T1082 K20  ; 爐體伺服機構無歸零要求
      MPP
      ANI     L3113  ; 出手臂取手歸零要求
      ANI     L3213  ; 出料托框昇降歸零要求
      ANI     L3313  ; 出左開夾歸零要求
      ANI     L3413  ; 出右開夾歸零要求
      ANI     L3513  ; 出板牙插移載歸零要求
      OUT     T1084 K20  ; 出料伺服機構無歸零要求
800   LD      SM400  ; Run On\
      MPS
      ANI     L1125  ; 整板    DO HOME
      ANI     L1225  ; 牙插移載DO HOME
      ANI     L1325  ; 備用 DO HOME
      ANI     L1425  ; 進手臂夾爪   DO HOME
      ANI     L1525  ; 進料托框昇降    DO HOME
      ANI     L1625  ; 進左開爪DO HOME
      ANI     L1725  ; 進右開爪DO HOME
      OUT     T1091 K20  ; 進料伺服機構無回原點訊號
      MRD
      ANI     L2125  ; 分流前取框   DO HOME
      ANI     L2225  ; 合流後掛框    DO HOME
      OUT     T1092 K20  ; 爐體伺服機構無回原點訊號
      MPP
      ANI     L3125  ; 出手臂夾爪   DO HOME
      ANI     L3225  ; 出料托框昇降    DO HOME
      ANI     L3325  ; 出左開夾DO HOME
      ANI     L3425  ; 出右開夾DO HOME
      ANI     L3525  ; 出板牙插移載    DO HOME
      OUT     T1094 K20  ; 出料伺服機構無回原點訊號
830   LD      SM400  ; Run On\
      MPS
      AND     T1081  ; 進料伺服機構無歸零要求
      AND     T1082  ; 爐體伺服機構無歸零要求
      AND     T1084  ; 出料伺服機構無歸零要求
      OUT     B32C1  ; 伺服機構無歸零要求
      MPP
      AND     T1091  ; 進料伺服機構無回原點訊號
      AND     T1092  ; 爐體伺服機構無回原點訊號
      AND     T1094  ; 出料伺服機構無回原點訊號
      OUT     B32C2  ; 伺服機構無回原點訊號
841   LD      M5531  ; 機台允許啟動
      OR      L3601  ; 停止中  信號
      AND     M3700  ; 啟動SW
      AND     B32C1  ; 伺服機構無歸零要求
      OUT     T900 K5  ; 啟動延遲
      AND     T900  ; 啟動延遲
      PLS     L3620  ; 啟動PLS
852   LD      M3701  ; 停止SW
      OUT     T901 K5  ; 停止延遲
      OUT     T909 K30  ; 強制停止延遲
861   LD      T901  ; 停止延遲
      MEP
      OR      L3601  ; 停止中  信號
      LDI     L3643  ; 進料手動信號
      ORI     L3648  ; 出料手動信號
      ANB
      AND     L3630  ; 啟動信號
      ANI     L3620  ; 啟動PLS
      OUT     L3601  ; 停止中  信號
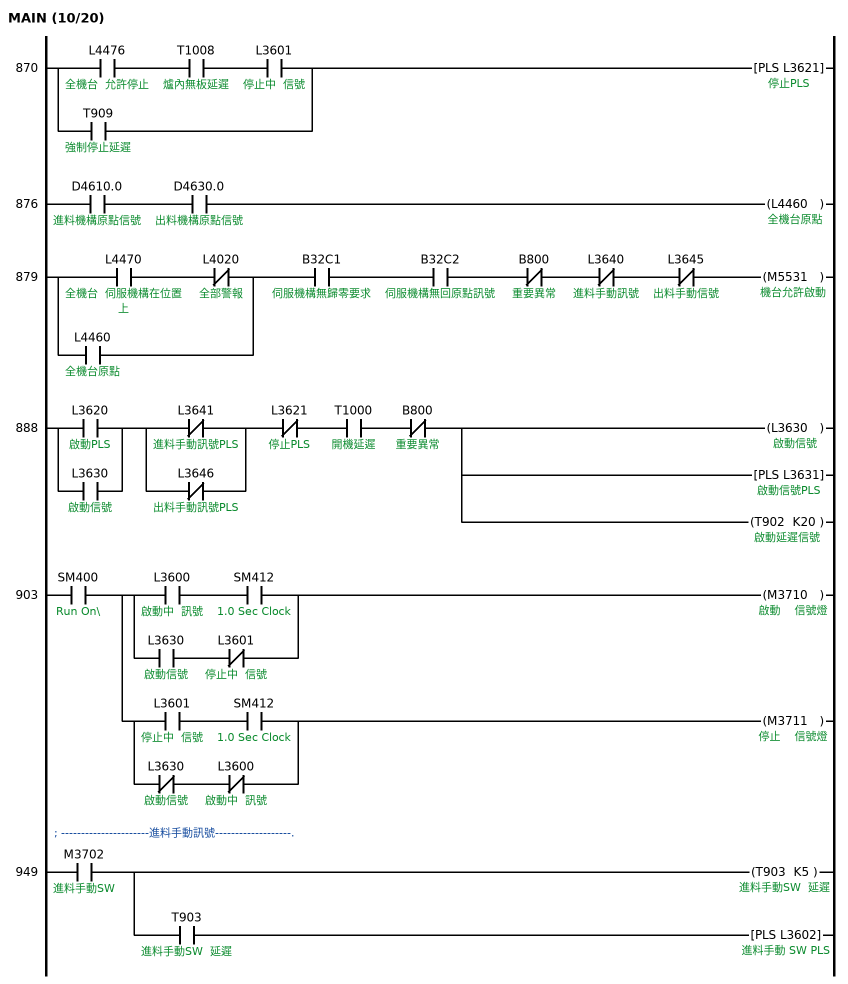
870   LD      L4476  ; 全機台  允許停止
      AND     T1008  ; 爐內無板延遲
      AND     L3601  ; 停止中  信號
      OR      T909  ; 強制停止延遲
      PLS     L3621  ; 停止PLS
876   LD      D4610.0  ; 進料機構原點信號
      AND     D4630.0  ; 出料機構原點信號
      OUT     L4460  ; 全機台原點
879   LD      L4470  ; 全機台  伺服機構在位置上
      ANI     L4020  ; 全部警報
      OR      L4460  ; 全機台原點
      AND     B32C1  ; 伺服機構無歸零要求
      AND     B32C2  ; 伺服機構無回原點訊號
      ANI     B800  ; 重要異常
      ANI     L3640  ; 進料手動訊號
      ANI     L3645  ; 出料手動信號
      OUT     M5531  ; 機台允許啟動
888   LD      L3620  ; 啟動PLS
      OR      L3630  ; 啟動信號
      LDI     L3641  ; 進料手動訊號PLS
      ORI     L3646  ; 出料手動訊號PLS
      ANB
      ANI     L3621  ; 停止PLS
      AND     T1000  ; 開機延遲
      ANI     B800  ; 重要異常
      OUT     L3630  ; 啟動信號
      PLS     L3631  ; 啟動信號PLS
      OUT     T902 K20  ; 啟動延遲信號
903   LD      SM400  ; Run On\
      MPS
      LD      L3600  ; 啟動中  訊號
      AND     SM412  ; 1.0 Sec Clock
      LD      L3630  ; 啟動信號
      ANI     L3601  ; 停止中  信號
      ORB
      ANB
      OUT     M3710  ; 啟動    信號燈
      MPP
      LD      L3601  ; 停止中  信號
      AND     SM412  ; 1.0 Sec Clock
      LDI     L3630  ; 啟動信號
      ANI     L3600  ; 啟動中  訊號
      ORB
      ANB
      OUT     M3711  ; 停止    信號燈
; ----------------------進料手動訊號-------------------.
949   LD      M3702  ; 進料手動SW
      OUT     T903 K5  ; 進料手動SW  延遲
      AND     T903  ; 進料手動SW  延遲
      PLS     L3602  ; 進料手動 SW PLS
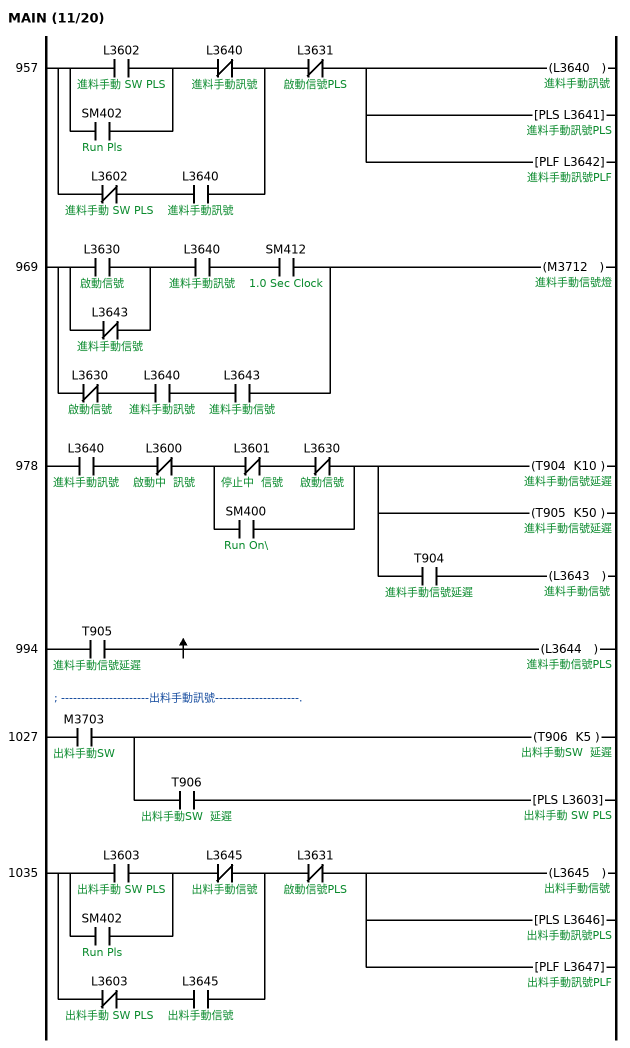
957   LD      L3602  ; 進料手動 SW PLS
      OR      SM402  ; Run Pls
      ANI     L3640  ; 進料手動訊號
      LDI     L3602  ; 進料手動 SW PLS
      AND     L3640  ; 進料手動訊號
      ORB
      ANI     L3631  ; 啟動信號PLS
      OUT     L3640  ; 進料手動訊號
      PLS     L3641  ; 進料手動訊號PLS
      PLF     L3642  ; 進料手動訊號PLF
969   LD      L3630  ; 啟動信號
      ORI     L3643  ; 進料手動信號
      AND     L3640  ; 進料手動訊號
      AND     SM412  ; 1.0 Sec Clock
      LDI     L3630  ; 啟動信號
      AND     L3640  ; 進料手動訊號
      AND     L3643  ; 進料手動信號
      ORB
      OUT     M3712  ; 進料手動信號燈
978   LD      L3640  ; 進料手動訊號
      ANI     L3600  ; 啟動中  訊號
      LDI     L3601  ; 停止中  信號
      ANI     L3630  ; 啟動信號
      OR      SM400  ; Run On\
      ANB
      OUT     T904 K10  ; 進料手動信號延遲
      OUT     T905 K50  ; 進料手動信號延遲
      AND     T904  ; 進料手動信號延遲
      OUT     L3643  ; 進料手動信號
994   LD      T905  ; 進料手動信號延遲
      MEP
      OUT     L3644  ; 進料手動信號PLS
; ----------------------出料手動訊號---------------------.
1027  LD      M3703  ; 出料手動SW
      OUT     T906 K5  ; 出料手動SW  延遲
      AND     T906  ; 出料手動SW  延遲
      PLS     L3603  ; 出料手動 SW PLS
1035  LD      L3603  ; 出料手動 SW PLS
      OR      SM402  ; Run Pls
      ANI     L3645  ; 出料手動信號
      LDI     L3603  ; 出料手動 SW PLS
      AND     L3645  ; 出料手動信號
      ORB
      ANI     L3631  ; 啟動信號PLS
      OUT     L3645  ; 出料手動信號
      PLS     L3646  ; 出料手動訊號PLS
      PLF     L3647  ; 出料手動訊號PLF
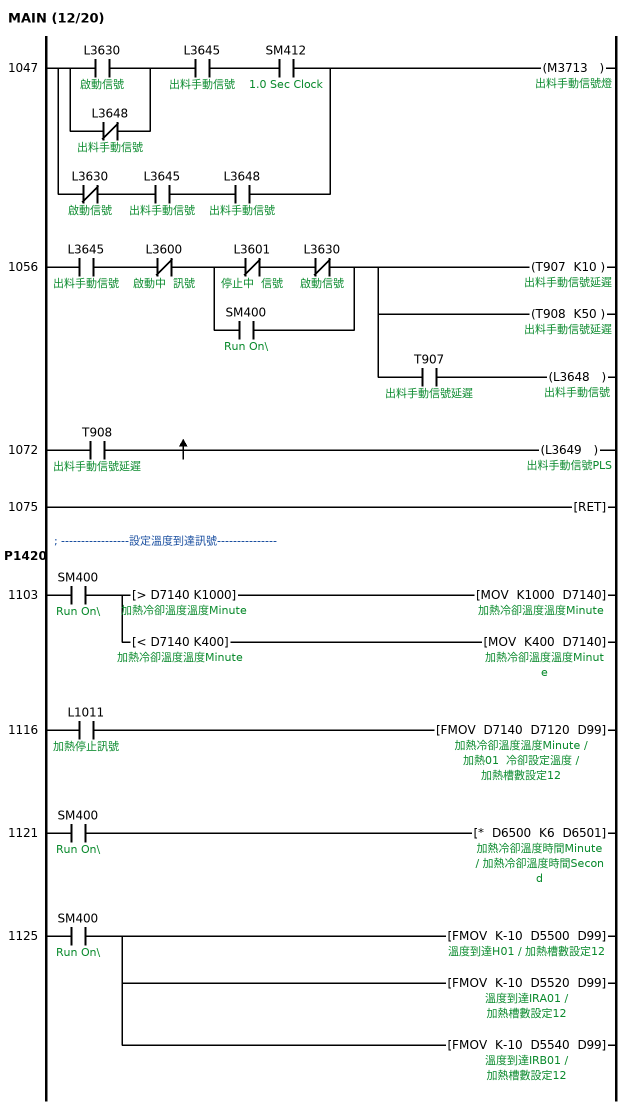
1047  LD      L3630  ; 啟動信號
      ORI     L3648  ; 出料手動信號
      AND     L3645  ; 出料手動信號
      AND     SM412  ; 1.0 Sec Clock
      LDI     L3630  ; 啟動信號
      AND     L3645  ; 出料手動信號
      AND     L3648  ; 出料手動信號
      ORB
      OUT     M3713  ; 出料手動信號燈
1056  LD      L3645  ; 出料手動信號
      ANI     L3600  ; 啟動中  訊號
      LDI     L3601  ; 停止中  信號
      ANI     L3630  ; 啟動信號
      OR      SM400  ; Run On\
      ANB
      OUT     T907 K10  ; 出料手動信號延遲
      OUT     T908 K50  ; 出料手動信號延遲
      AND     T907  ; 出料手動信號延遲
      OUT     L3648  ; 出料手動信號
1072  LD      T908  ; 出料手動信號延遲
      MEP
      OUT     L3649  ; 出料手動信號PLS
1075  RET
; -----------------設定溫度到達訊號---------------
      P1420
1103  LD      SM400  ; Run On\
      MPS
      AND>    D7140 K1000  ; 加熱冷卻溫度溫度Minute
      MOV     K1000 D7140
      MPP
      AND<    D7140 K400  ; 加熱冷卻溫度溫度Minute
      MOV     K400 D7140
1116  LD      L1011  ; 加熱停止訊號
      FMOV    D7140 D7120 D99  ; 加熱01  冷卻設定溫度
1121  LD      SM400  ; Run On\
      *       D6500 K6 D6501  ; 加熱冷卻溫度時間Minute / 加熱冷卻溫度時間Second
1125  LD      SM400  ; Run On\
      FMOV    K-10 D5500 D99  ; 溫度到達H01
      FMOV    K-10 D5520 D99  ; 溫度到達IRA01
      FMOV    K-10 D5540 D99  ; 溫度到達IRB01
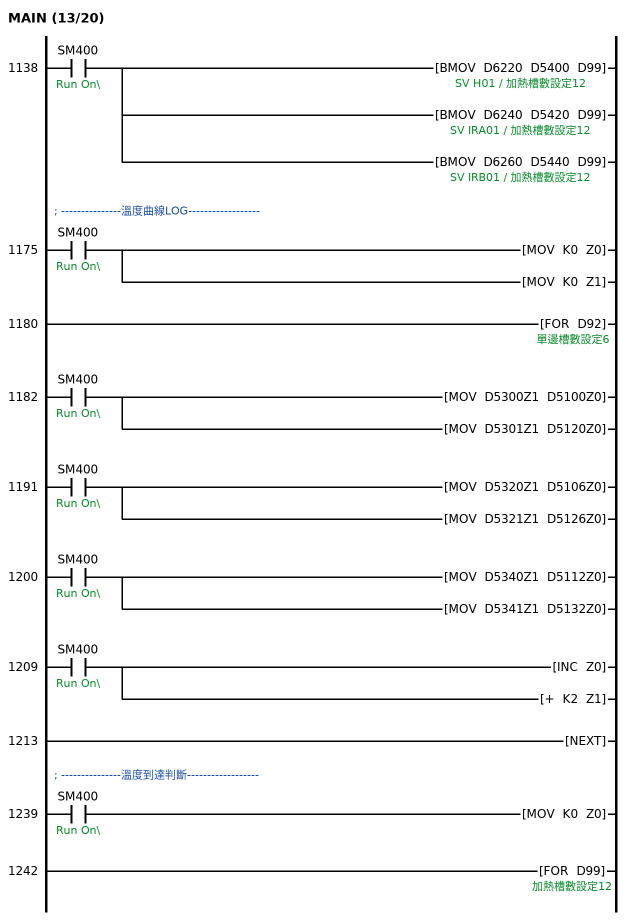
1138  LD      SM400  ; Run On\
      BMOV    D6220 D5400 D99  ; SV H01
      BMOV    D6240 D5420 D99  ; SV IRA01
      BMOV    D6260 D5440 D99  ; SV IRB01
; ---------------溫度曲線LOG------------------
1175  LD      SM400  ; Run On\
      MOV     K0 Z0
      MOV     K0 Z1
1180  FOR     D92
1182  LD      SM400  ; Run On\
      MOV     D5300Z1 D5100Z0
      MOV     D5301Z1 D5120Z0
1191  LD      SM400  ; Run On\
      MOV     D5320Z1 D5106Z0
      MOV     D5321Z1 D5126Z0
1200  LD      SM400  ; Run On\
      MOV     D5340Z1 D5112Z0
      MOV     D5341Z1 D5132Z0
1209  LD      SM400  ; Run On\
      INC     Z0
      +       K2 Z1
1213  NEXT
; ---------------溫度到達判斷------------------
1239  LD      SM400  ; Run On\
      MOV     K0 Z0
1242  FOR     D99
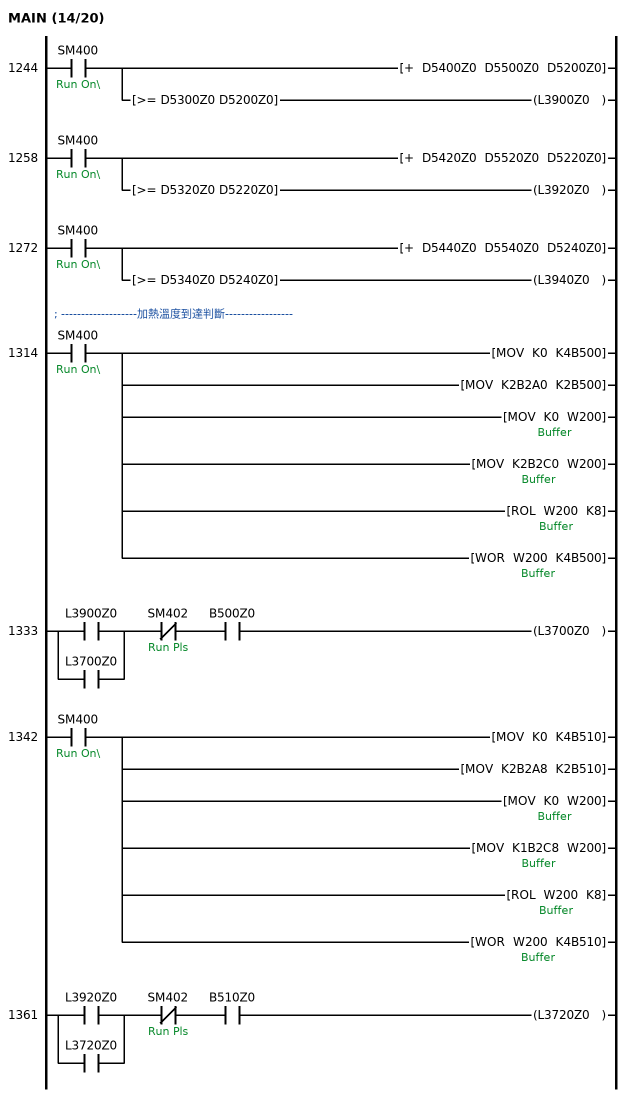
1244  LD      SM400  ; Run On\
      +       D5400Z0 D5500Z0 D5200Z0
      AND>=   D5300Z0 D5200Z0
      OUT     L3900Z0
1258  LD      SM400  ; Run On\
      +       D5420Z0 D5520Z0 D5220Z0
      AND>=   D5320Z0 D5220Z0
      OUT     L3920Z0
1272  LD      SM400  ; Run On\
      +       D5440Z0 D5540Z0 D5240Z0
      AND>=   D5340Z0 D5240Z0
      OUT     L3940Z0
; -------------------加熱溫度到達判斷-----------------
1314  LD      SM400  ; Run On\
      MOV     K0 K4B500  ; 第01槽  熱風電磁開關
      MOV     K2B2A0 K2B500  ; 第01槽熱風H01電磁開關
      MOV     K0 W200  ; Buffer
      MOV     K2B2C0 W200  ; 第09槽熱風H09電磁開關
      ROL     W200 K8
      WOR     W200 K4B500
1333  LD      L3900Z0
      OR      L3700Z0
      ANI     SM402  ; Run Pls
      AND     B500Z0
      OUT     L3700Z0
1342  LD      SM400  ; Run On\
      MOV     K0 K4B510  ; 第01槽  IRA 電磁開關
      MOV     K2B2A8 K2B510  ; 第01槽IR01A電磁開關
      MOV     K0 W200
      MOV     K1B2C8 W200  ; 第09槽IR09A電磁開關
      ROL     W200 K8
      WOR     W200 K4B510
1361  LD      L3920Z0
      OR      L3720Z0
      ANI     SM402  ; Run Pls
      AND     B510Z0
      OUT     L3720Z0
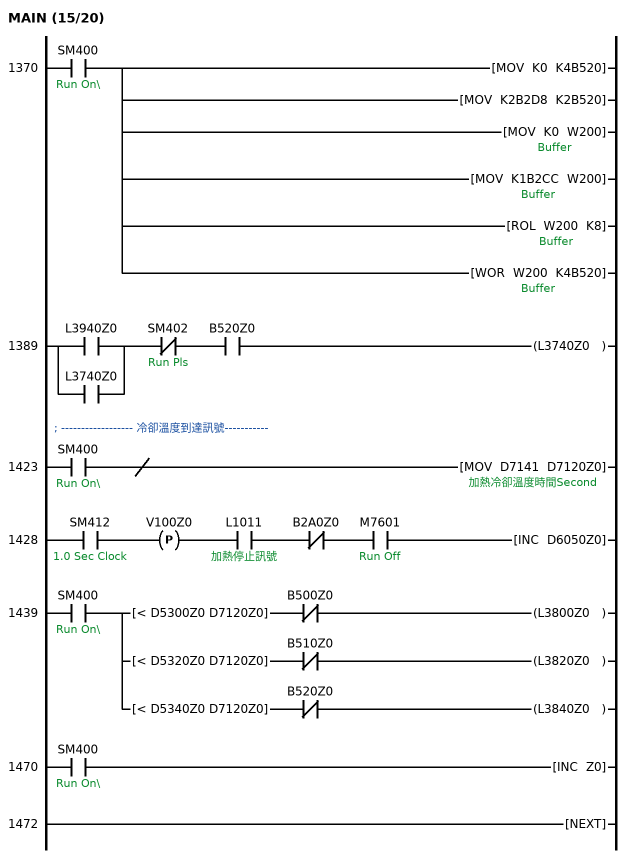
1370  LD      SM400  ; Run On\
      MOV     K0 K4B520  ; 第01槽  IRB 電磁開關
      MOV     K2B2D8 K2B520  ; 第01槽IR01B電磁開關
      MOV     K0 W200
      MOV     K1B2CC W200  ; 第09槽IR09B電磁開關
      ROL     W200 K8
      WOR     W200 K4B520
1389  LD      L3940Z0
      OR      L3740Z0
      ANI     SM402  ; Run Pls
      AND     B520Z0
      OUT     L3740Z0
; ------------------ 冷卻溫度到達訊號-----------
1423  LD      SM400  ; Run On\
      INV
      MOV     D7141 D7120Z0  ; 加熱冷卻溫度時間Second
1428  LD      SM412  ; 1.0 Sec Clock
      EGP     V100Z0
      AND     L1011  ; 加熱停止訊號
      ANI     B2A0Z0
      AND     M7601  ; Run Off
      INC     D6050Z0
1439  LD      SM400  ; Run On\
      MPS
      AND<    D5300Z0 D7120Z0
      ANI     B500Z0
      OUT     L3800Z0
      MRD
      AND<    D5320Z0 D7120Z0
      ANI     B510Z0
      OUT     L3820Z0
      MPP
      AND<    D5340Z0 D7120Z0
      ANI     B520Z0
      OUT     L3840Z0
1470  LD      SM400  ; Run On\
      INC     Z0
1472  NEXT
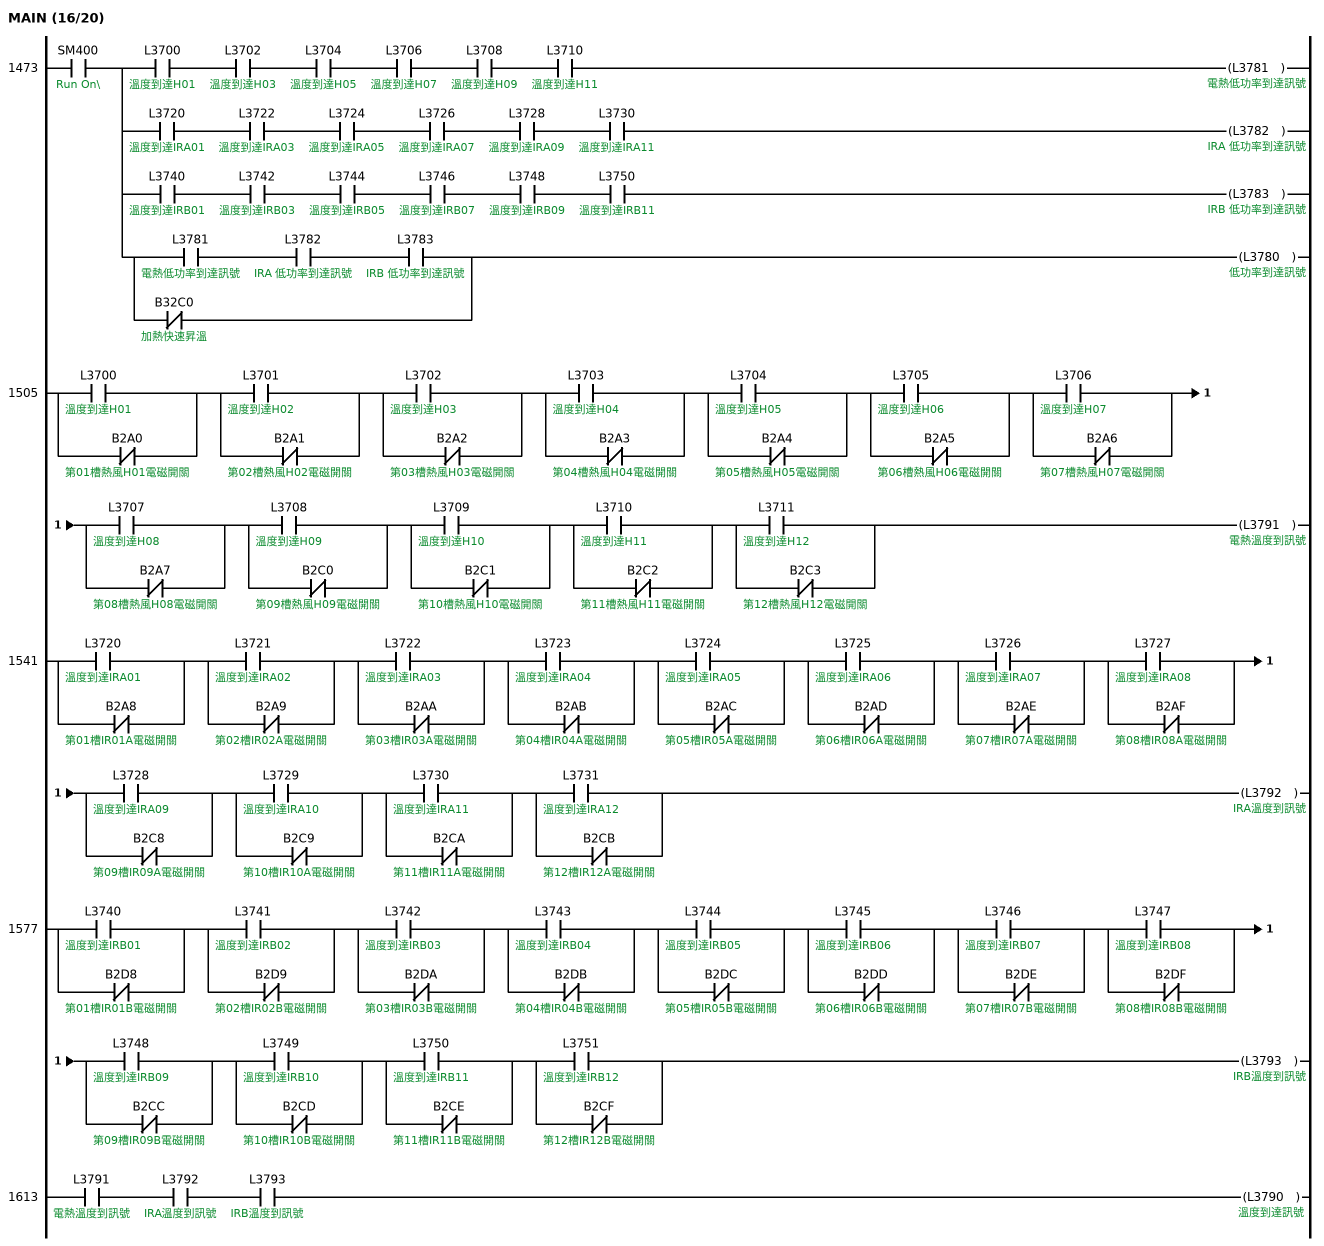
1473  LD      SM400  ; Run On\
      MPS
      AND     L3700  ; 溫度到達H01
      AND     L3702  ; 溫度到達H03
      AND     L3704  ; 溫度到達H05
      AND     L3706  ; 溫度到達H07
      AND     L3708  ; 溫度到達H09
      AND     L3710  ; 溫度到達H11
      OUT     L3781  ; 電熱低功率到達訊號
      MRD
      AND     L3720  ; 溫度到達IRA01
      AND     L3722  ; 溫度到達IRA03
      AND     L3724  ; 溫度到達IRA05
      AND     L3726  ; 溫度到達IRA07
      AND     L3728  ; 溫度到達IRA09
      AND     L3730  ; 溫度到達IRA11
      OUT     L3782  ; IRA 低功率到達訊號
      MRD
      AND     L3740  ; 溫度到達IRB01
      AND     L3742  ; 溫度到達IRB03
      AND     L3744  ; 溫度到達IRB05
      AND     L3746  ; 溫度到達IRB07
      AND     L3748  ; 溫度到達IRB09
      AND     L3750  ; 溫度到達IRB11
      OUT     L3783  ; IRB 低功率到達訊號
      MPP
      LD      L3781  ; 電熱低功率到達訊號
      AND     L3782  ; IRA 低功率到達訊號
      AND     L3783  ; IRB 低功率到達訊號
      ORI     B32C0  ; 加熱快速昇溫
      ANB
      OUT     L3780  ; 低功率到達訊號
1505  LD      L3700  ; 溫度到達H01
      ORI     B2A0  ; 第01槽熱風H01電磁開關
      LD      L3701  ; 溫度到達H02
      ORI     B2A1  ; 第02槽熱風H02電磁開關
      ANB
      LD      L3702  ; 溫度到達H03
      ORI     B2A2  ; 第03槽熱風H03電磁開關
      ANB
      LD      L3703  ; 溫度到達H04
      ORI     B2A3  ; 第04槽熱風H04電磁開關
      ANB
      LD      L3704  ; 溫度到達H05
      ORI     B2A4  ; 第05槽熱風H05電磁開關
      ANB
      LD      L3705  ; 溫度到達H06
      ORI     B2A5  ; 第06槽熱風H06電磁開關
      ANB
      LD      L3706  ; 溫度到達H07
      ORI     B2A6  ; 第07槽熱風H07電磁開關
      ANB
      LD      L3707  ; 溫度到達H08
      ORI     B2A7  ; 第08槽熱風H08電磁開關
      ANB
      LD      L3708  ; 溫度到達H09
      ORI     B2C0  ; 第09槽熱風H09電磁開關
      ANB
      LD      L3709  ; 溫度到達H10
      ORI     B2C1  ; 第10槽熱風H10電磁開關
      ANB
      LD      L3710  ; 溫度到達H11
      ORI     B2C2  ; 第11槽熱風H11電磁開關
      ANB
      LD      L3711  ; 溫度到達H12
      ORI     B2C3  ; 第12槽熱風H12電磁開關
      ANB
      OUT     L3791  ; 電熱溫度到訊號
1541  LD      L3720  ; 溫度到達IRA01
      ORI     B2A8  ; 第01槽IR01A電磁開關
      LD      L3721  ; 溫度到達IRA02
      ORI     B2A9  ; 第02槽IR02A電磁開關
      ANB
      LD      L3722  ; 溫度到達IRA03
      ORI     B2AA  ; 第03槽IR03A電磁開關
      ANB
      LD      L3723  ; 溫度到達IRA04
      ORI     B2AB  ; 第04槽IR04A電磁開關
      ANB
      LD      L3724  ; 溫度到達IRA05
      ORI     B2AC  ; 第05槽IR05A電磁開關
      ANB
      LD      L3725  ; 溫度到達IRA06
      ORI     B2AD  ; 第06槽IR06A電磁開關
      ANB
      LD      L3726  ; 溫度到達IRA07
      ORI     B2AE  ; 第07槽IR07A電磁開關
      ANB
      LD      L3727  ; 溫度到達IRA08
      ORI     B2AF  ; 第08槽IR08A電磁開關
      ANB
      LD      L3728  ; 溫度到達IRA09
      ORI     B2C8  ; 第09槽IR09A電磁開關
      ANB
      LD      L3729  ; 溫度到達IRA10
      ORI     B2C9  ; 第10槽IR10A電磁開關
      ANB
      LD      L3730  ; 溫度到達IRA11
      ORI     B2CA  ; 第11槽IR11A電磁開關
      ANB
      LD      L3731  ; 溫度到達IRA12
      ORI     B2CB  ; 第12槽IR12A電磁開關
      ANB
      OUT     L3792  ; IRA溫度到訊號
1577  LD      L3740  ; 溫度到達IRB01
      ORI     B2D8  ; 第01槽IR01B電磁開關
      LD      L3741  ; 溫度到達IRB02
      ORI     B2D9  ; 第02槽IR02B電磁開關
      ANB
      LD      L3742  ; 溫度到達IRB03
      ORI     B2DA  ; 第03槽IR03B電磁開關
      ANB
      LD      L3743  ; 溫度到達IRB04
      ORI     B2DB  ; 第04槽IR04B電磁開關
      ANB
      LD      L3744  ; 溫度到達IRB05
      ORI     B2DC  ; 第05槽IR05B電磁開關
      ANB
      LD      L3745  ; 溫度到達IRB06
      ORI     B2DD  ; 第06槽IR06B電磁開關
      ANB
      LD      L3746  ; 溫度到達IRB07
      ORI     B2DE  ; 第07槽IR07B電磁開關
      ANB
      LD      L3747  ; 溫度到達IRB08
      ORI     B2DF  ; 第08槽IR08B電磁開關
      ANB
      LD      L3748  ; 溫度到達IRB09
      ORI     B2CC  ; 第09槽IR09B電磁開關
      ANB
      LD      L3749  ; 溫度到達IRB10
      ORI     B2CD  ; 第10槽IR10B電磁開關
      ANB
      LD      L3750  ; 溫度到達IRB11
      ORI     B2CE  ; 第11槽IR11B電磁開關
      ANB
      LD      L3751  ; 溫度到達IRB12
      ORI     B2CF  ; 第12槽IR12B電磁開關
      ANB
      OUT     L3793  ; IRB溫度到訊號
1613  LD      L3791  ; 電熱溫度到訊號
      AND     L3792  ; IRA溫度到訊號
      AND     L3793  ; IRB溫度到訊號
      OUT     L3790  ; 溫度到達訊號
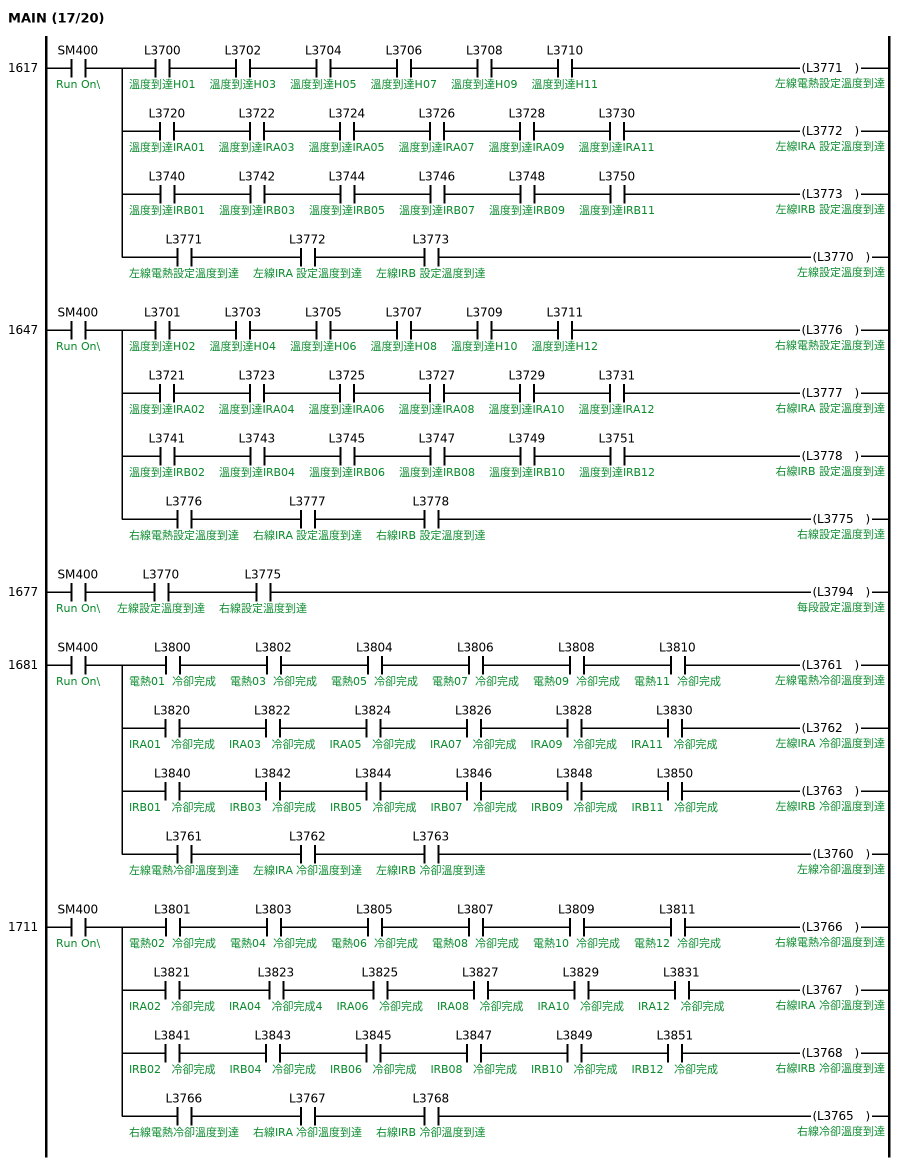
1617  LD      SM400  ; Run On\
      MPS
      AND     L3700  ; 溫度到達H01
      AND     L3702  ; 溫度到達H03
      AND     L3704  ; 溫度到達H05
      AND     L3706  ; 溫度到達H07
      AND     L3708  ; 溫度到達H09
      AND     L3710  ; 溫度到達H11
      OUT     L3771  ; 左線電熱設定溫度到達
      MRD
      AND     L3720  ; 溫度到達IRA01
      AND     L3722  ; 溫度到達IRA03
      AND     L3724  ; 溫度到達IRA05
      AND     L3726  ; 溫度到達IRA07
      AND     L3728  ; 溫度到達IRA09
      AND     L3730  ; 溫度到達IRA11
      OUT     L3772  ; 左線IRA 設定溫度到達
      MRD
      AND     L3740  ; 溫度到達IRB01
      AND     L3742  ; 溫度到達IRB03
      AND     L3744  ; 溫度到達IRB05
      AND     L3746  ; 溫度到達IRB07
      AND     L3748  ; 溫度到達IRB09
      AND     L3750  ; 溫度到達IRB11
      OUT     L3773  ; 左線IRB 設定溫度到達
      MPP
      AND     L3771  ; 左線電熱設定溫度到達
      AND     L3772  ; 左線IRA 設定溫度到達
      AND     L3773  ; 左線IRB 設定溫度到達
      OUT     L3770  ; 左線設定溫度到達
1647  LD      SM400  ; Run On\
      MPS
      AND     L3701  ; 溫度到達H02
      AND     L3703  ; 溫度到達H04
      AND     L3705  ; 溫度到達H06
      AND     L3707  ; 溫度到達H08
      AND     L3709  ; 溫度到達H10
      AND     L3711  ; 溫度到達H12
      OUT     L3776  ; 右線電熱設定溫度到達
      MRD
      AND     L3721  ; 溫度到達IRA02
      AND     L3723  ; 溫度到達IRA04
      AND     L3725  ; 溫度到達IRA06
      AND     L3727  ; 溫度到達IRA08
      AND     L3729  ; 溫度到達IRA10
      AND     L3731  ; 溫度到達IRA12
      OUT     L3777  ; 右線IRA 設定溫度到達
      MRD
      AND     L3741  ; 溫度到達IRB02
      AND     L3743  ; 溫度到達IRB04
      AND     L3745  ; 溫度到達IRB06
      AND     L3747  ; 溫度到達IRB08
      AND     L3749  ; 溫度到達IRB10
      AND     L3751  ; 溫度到達IRB12
      OUT     L3778  ; 右線IRB 設定溫度到達
      MPP
      AND     L3776  ; 右線電熱設定溫度到達
      AND     L3777  ; 右線IRA 設定溫度到達
      AND     L3778  ; 右線IRB 設定溫度到達
      OUT     L3775  ; 右線設定溫度到達
1677  LD      SM400  ; Run On\
      AND     L3770  ; 左線設定溫度到達
      AND     L3775  ; 右線設定溫度到達
      OUT     L3794  ; 每段設定溫度到達
1681  LD      SM400  ; Run On\
      MPS
      AND     L3800  ; 電熱01  冷卻完成
      AND     L3802  ; 電熱03  冷卻完成
      AND     L3804  ; 電熱05  冷卻完成
      AND     L3806  ; 電熱07  冷卻完成
      AND     L3808  ; 電熱09  冷卻完成
      AND     L3810  ; 電熱11  冷卻完成
      OUT     L3761  ; 左線電熱冷卻溫度到達
      MRD
      AND     L3820  ; IRA01   冷卻完成
      AND     L3822  ; IRA03   冷卻完成
      AND     L3824  ; IRA05   冷卻完成
      AND     L3826  ; IRA07   冷卻完成
      AND     L3828  ; IRA09   冷卻完成
      AND     L3830  ; IRA11   冷卻完成
      OUT     L3762  ; 左線IRA 冷卻溫度到達
      MRD
      AND     L3840  ; IRB01   冷卻完成
      AND     L3842  ; IRB03   冷卻完成
      AND     L3844  ; IRB05   冷卻完成
      AND     L3846  ; IRB07   冷卻完成
      AND     L3848  ; IRB09   冷卻完成
      AND     L3850  ; IRB11   冷卻完成
      OUT     L3763  ; 左線IRB 冷卻溫度到達
      MPP
      AND     L3761  ; 左線電熱冷卻溫度到達
      AND     L3762  ; 左線IRA 冷卻溫度到達
      AND     L3763  ; 左線IRB 冷卻溫度到達
      OUT     L3760  ; 左線冷卻溫度到達
1711  LD      SM400  ; Run On\
      MPS
      AND     L3801  ; 電熱02  冷卻完成
      AND     L3803  ; 電熱04  冷卻完成
      AND     L3805  ; 電熱06  冷卻完成
      AND     L3807  ; 電熱08  冷卻完成
      AND     L3809  ; 電熱10  冷卻完成
      AND     L3811  ; 電熱12  冷卻完成
      OUT     L3766  ; 右線電熱冷卻溫度到達
      MRD
      AND     L3821  ; IRA02   冷卻完成
      AND     L3823  ; IRA04   冷卻完成4
      AND     L3825  ; IRA06   冷卻完成
      AND     L3827  ; IRA08   冷卻完成
      AND     L3829  ; IRA10   冷卻完成
      AND     L3831  ; IRA12   冷卻完成
      OUT     L3767  ; 右線IRA 冷卻溫度到達
      MRD
      AND     L3841  ; IRB02   冷卻完成
      AND     L3843  ; IRB04   冷卻完成
      AND     L3845  ; IRB06   冷卻完成
      AND     L3847  ; IRB08   冷卻完成
      AND     L3849  ; IRB10   冷卻完成
      AND     L3851  ; IRB12   冷卻完成
      OUT     L3768  ; 右線IRB 冷卻溫度到達
      MPP
      AND     L3766  ; 右線電熱冷卻溫度到達
      AND     L3767  ; 右線IRA 冷卻溫度到達
      AND     L3768  ; 右線IRB 冷卻溫度到達
      OUT     L3765  ; 右線冷卻溫度到達
